SPLINE
SPL {X  -157.536, Y  +349.586, Z    +0.000, E1   +71.787, E3 +25840.740}
SPL {X  -154.855, Y  +337.291, Z    +0.000, E1   +72.155, E3 +25845.494}
SPL {X  -150.925, Y  +324.412, Z    +0.000, E1   +72.419, E3 +25851.389}
SPL {X  -146.819, Y  +313.931, Z    +0.000, E1   +72.621, E3 +25856.082}
SPL {X  -140.820, Y  +301.561, Z    +0.000, E1   +73.023, E3 +25859.998}
SPL {X  -136.475, Y  +294.006, Z    +0.000, E1   +72.670, E3 +25866.907}
SPL {X  -133.214, Y  +288.895, Z    +0.000, E1   +72.272, E3 +25872.555}
SPL {X  -129.829, Y  +284.006, Z    +0.000, E1   +71.844, E3 +25878.030}
SPL {X  -126.314, Y  +279.309, Z    +0.000, E1   +71.374, E3 +25883.322}
SPL {X  -122.705, Y  +274.834, Z    +0.000, E1   +70.869, E3 +25888.333}
SPL {X  -119.804, Y  +271.463, Z    +0.000, E1   +70.429, E3 +25892.052}
SPL {X   -77.409, Y  +237.483, Z    +0.000, E1   +59.013, E3 +25985.728}
ENDSPLINE

SPLINE
SPL {X  -103.775, Y  +255.731, Z    +0.000, E1   +56.205, E3 +26182.441}
SPL {X  -141.196, Y  +302.265, Z    +0.000, E1   +49.914, E3 +26219.926}
SPL {X  -155.405, Y  +339.473, Z    +0.000, E1   +34.418, E3 +26229.626}
SPL {X  -159.172, Y  +361.346, Z    +0.000, E1   +18.323, E3 +26232.051}
SPL {X  -159.962, Y  +374.520, Z    +0.000, E1    +5.534, E3 +26232.664}
SPL {X  -159.990, Y  +379.490, Z    +0.000, E1    +0.023, E3 +26232.721}
SPL {X  -159.990, Y  +381.667, Z    +0.000, E1    -4.707, E3 +26232.743}
SPL {X  -159.990, Y  +387.434, Z    +0.000, E1   -19.600, E3 +26232.926}
SPL {X  -159.990, Y  +395.000, Z    +0.000, E1   -38.121, E3 +26233.435}
SPL {X  -159.990, Y  +406.380, Z    +0.000, E1   -55.108, E3 +26234.876}
SPL {X  -159.990, Y  +426.664, Z    +0.000, E1   -66.963, E3 +26239.066}
SPL {X  -159.990, Y  +494.829, Z    +0.000, E1   -73.764, E3 +26260.831}
SPL {X  -158.798, Y  +695.991, Z    +0.000, E1   -74.986, E3 +26350.763}
SPL {X  -156.512, Y  +709.677, Z    +0.000, E1   -74.772, E3 +26360.907}
SPL {X  -153.684, Y  +720.975, Z    +0.000, E1   -74.508, E3 +26370.194}
SPL {X  -149.353, Y  +733.863, Z    +0.000, E1   -74.100, E3 +26381.782}
SPL {X  -145.190, Y  +743.705, Z    +0.000, E1   -73.640, E3 +26391.463}
SPL {X  -141.940, Y  +750.322, Z    +0.000, E1   -73.290, E3 +26398.230}
SPL {X  -138.555, Y  +756.496, Z    +0.000, E1   -72.905, E3 +26404.795}
SPL {X  -135.025, Y  +762.319, Z    +0.000, E1   -72.483, E3 +26411.174}
SPL {X  -131.747, Y  +767.272, Z    +0.000, E1   -72.071, E3 +26416.699}
SPL {X  -127.432, Y  +773.236, Z    +0.000, E1   -71.530, E3 +26423.385}
SPL {X  -124.036, Y  +777.554, Z    +0.000, E1   -71.026, E3 +26428.283}
SPL {X  -120.782, Y  +781.422, Z    +0.000, E1   -70.584, E3 +26432.541}
SPL {X   -74.295, Y  +818.193, Z    +0.000, E1   -57.793, E3 +26542.872}
ENDSPLINE

SPLINE
SPL {X  -105.102, Y  +797.125, Z    +0.000, E1   -55.734, E3 +26722.238}
SPL {X  -126.361, Y  +774.631, Z    +0.000, E1   -54.192, E3 +26747.906}
SPL {X  -145.777, Y  +742.423, Z    +0.000, E1   -46.722, E3 +26763.247}
SPL {X  -154.920, Y  +716.458, Z    +0.000, E1   -35.175, E3 +26769.302}
SPL {X  -159.063, Y  +693.702, Z    +0.000, E1   -19.028, E3 +26772.083}
SPL {X  -159.958, Y  +679.684, Z    +0.000, E1    -5.688, E3 +26772.795}
SPL {X  -159.990, Y  +674.512, Z    +0.000, E1    -0.026, E3 +26772.860}
SPL {X  -159.990, Y  +672.767, Z    +0.000, E1    +3.705, E3 +26772.873}
SPL {X  -159.990, Y  +669.310, Z    +0.000, E1   +12.444, E3 +26772.947}
SPL {X  -159.990, Y  +665.511, Z    +0.000, E1   +22.359, E3 +26773.106}
SPL {X  -159.990, Y  +660.776, Z    +0.000, E1   +34.018, E3 +26773.413}
SPL {X  -159.990, Y  +655.863, Z    +0.000, E1   +43.768, E3 +26773.870}
SPL {X  -159.990, Y  +646.280, Z    +0.000, E1   +56.156, E3 +26775.159}
SPL {X  -159.990, Y  +625.549, Z    +0.000, E1   +67.208, E3 +26779.681}
SPL {X  -159.990, Y  +550.186, Z    +0.000, E1   +73.637, E3 +26805.087}
SPL {X  -159.493, Y  +364.902, Z    +0.000, E1   +74.541, E3 +26892.080}
SPL {X  -156.915, Y  +346.281, Z    +0.000, E1   +74.304, E3 +26905.676}
ENDSPLINE

SPLINE
SPL {X  -159.697, Y  +367.814, Z    +0.000, E1   +71.217, E3 +26922.994}
ENDSPLINE

SPLINE
SPL {X  -157.536, Y  +349.586, Z    +0.000, E1   +71.787, E3 +26930.293}
SPL {X  -154.855, Y  +337.291, Z    +0.000, E1   +72.155, E3 +26935.047}
SPL {X  -150.925, Y  +324.412, Z    +0.000, E1   +72.419, E3 +26940.941}
SPL {X  -146.819, Y  +313.931, Z    +0.000, E1   +72.621, E3 +26945.634}
SPL {X  -140.820, Y  +301.561, Z    +0.000, E1   +73.023, E3 +26949.550}
SPL {X  -136.475, Y  +294.006, Z    +0.000, E1   +72.670, E3 +26956.459}
SPL {X  -133.214, Y  +288.895, Z    +0.000, E1   +72.272, E3 +26962.107}
SPL {X  -129.829, Y  +284.006, Z    +0.000, E1   +71.844, E3 +26967.582}
SPL {X  -126.314, Y  +279.309, Z    +0.000, E1   +71.374, E3 +26972.874}
SPL {X  -122.705, Y  +274.834, Z    +0.000, E1   +70.869, E3 +26977.886}
SPL {X  -119.804, Y  +271.463, Z    +0.000, E1   +70.429, E3 +26981.604}
SPL {X   -77.409, Y  +237.483, Z    +0.000, E1   +59.013, E3 +27075.280}
ENDSPLINE

SPLINE
SPL {X  -103.775, Y  +255.731, Z    +0.000, E1   +56.205, E3 +27271.993}
SPL {X  -141.196, Y  +302.265, Z    +0.000, E1   +49.914, E3 +27309.478}
SPL {X  -155.405, Y  +339.473, Z    +0.000, E1   +34.418, E3 +27319.179}
SPL {X  -159.172, Y  +361.346, Z    +0.000, E1   +18.323, E3 +27321.603}
SPL {X  -159.962, Y  +374.520, Z    +0.000, E1    +5.534, E3 +27322.216}
SPL {X  -159.990, Y  +379.490, Z    +0.000, E1    +0.023, E3 +27322.274}
SPL {X  -159.990, Y  +381.667, Z    +0.000, E1    -4.707, E3 +27322.295}
SPL {X  -159.990, Y  +387.434, Z    +0.000, E1   -19.600, E3 +27322.478}
SPL {X  -159.990, Y  +395.000, Z    +0.000, E1   -38.121, E3 +27322.987}
SPL {X  -159.990, Y  +406.380, Z    +0.000, E1   -55.108, E3 +27324.429}
SPL {X  -159.990, Y  +426.664, Z    +0.000, E1   -66.963, E3 +27328.619}
SPL {X  -159.990, Y  +494.829, Z    +0.000, E1   -73.764, E3 +27350.383}
SPL {X  -158.798, Y  +695.991, Z    +0.000, E1   -74.986, E3 +27440.315}
SPL {X  -156.512, Y  +709.677, Z    +0.000, E1   -74.772, E3 +27450.459}
SPL {X  -153.684, Y  +720.975, Z    +0.000, E1   -74.508, E3 +27459.746}
SPL {X  -149.353, Y  +733.863, Z    +0.000, E1   -74.100, E3 +27471.334}
SPL {X  -145.190, Y  +743.705, Z    +0.000, E1   -73.640, E3 +27481.015}
SPL {X  -141.940, Y  +750.322, Z    +0.000, E1   -73.290, E3 +27487.782}
SPL {X  -138.555, Y  +756.496, Z    +0.000, E1   -72.905, E3 +27494.347}
SPL {X  -135.025, Y  +762.319, Z    +0.000, E1   -72.483, E3 +27500.727}
SPL {X  -131.747, Y  +767.272, Z    +0.000, E1   -72.071, E3 +27506.252}
SPL {X  -127.432, Y  +773.236, Z    +0.000, E1   -71.530, E3 +27512.937}
SPL {X  -124.036, Y  +777.554, Z    +0.000, E1   -71.026, E3 +27517.835}
SPL {X  -120.782, Y  +781.422, Z    +0.000, E1   -70.584, E3 +27522.093}
SPL {X   -74.295, Y  +818.193, Z    +0.000, E1   -57.793, E3 +27632.424}
ENDSPLINE

SPLINE
SPL {X  -105.102, Y  +797.125, Z    +0.000, E1   -55.734, E3 +27811.791}
SPL {X  -126.361, Y  +774.631, Z    +0.000, E1   -54.192, E3 +27837.458}
SPL {X  -145.777, Y  +742.423, Z    +0.000, E1   -46.722, E3 +27852.799}
SPL {X  -154.920, Y  +716.458, Z    +0.000, E1   -35.175, E3 +27858.854}
SPL {X  -158.252, Y  +700.019, Z    +0.000, E1   -24.087, E3 +27861.106}
SPL {X  -159.434, Y  +689.826, Z    +0.000, E1   -15.506, E3 +27861.924}
SPL {X  -159.958, Y  +679.684, Z    +0.000, E1    -5.688, E3 +27862.347}
SPL {X  -159.990, Y  +674.512, Z    +0.000, E1    -0.026, E3 +27862.412}
SPL {X  -159.990, Y  +672.767, Z    +0.000, E1    +3.705, E3 +27862.425}
SPL {X  -159.990, Y  +669.310, Z    +0.000, E1   +12.444, E3 +27862.499}
SPL {X  -159.990, Y  +665.511, Z    +0.000, E1   +22.359, E3 +27862.658}
SPL {X  -159.990, Y  +660.776, Z    +0.000, E1   +34.018, E3 +27862.965}
SPL {X  -159.990, Y  +655.863, Z    +0.000, E1   +43.768, E3 +27863.422}
SPL {X  -159.990, Y  +646.280, Z    +0.000, E1   +56.156, E3 +27864.712}
SPL {X  -159.990, Y  +625.549, Z    +0.000, E1   +67.208, E3 +27869.233}
SPL {X  -159.990, Y  +550.186, Z    +0.000, E1   +73.637, E3 +27894.639}
SPL {X  -159.878, Y  +371.520, Z    +0.000, E1   +74.559, E3 +27977.401}
SPL {X  -159.109, Y  +360.737, Z    +0.000, E1   +74.490, E3 +27984.525}
SPL {X  -156.915, Y  +346.281, Z    +0.000, E1   +74.304, E3 +27995.228}
ENDSPLINE

SPLINE
SPL {X  -159.697, Y  +367.814, Z    +0.000, E1   +71.217, E3 +28012.547}
ENDSPLINE

SPLINE
SPL {X  -156.028, Y  +342.114, Z    +0.000, E1   +72.020, E3 +28022.700}
SPL {X  -150.925, Y  +324.412, Z    +0.000, E1   +72.419, E3 +28030.493}
SPL {X  -144.972, Y  +309.824, Z    +0.000, E1   +72.799, E3 +28036.095}
SPL {X  -139.605, Y  +299.351, Z    +0.000, E1   +73.035, E3 +28040.227}
SPL {X  -136.475, Y  +294.006, Z    +0.000, E1   +72.670, E3 +28046.012}
SPL {X  -133.214, Y  +288.895, Z    +0.000, E1   +72.272, E3 +28051.659}
SPL {X  -129.829, Y  +284.006, Z    +0.000, E1   +71.844, E3 +28057.134}
SPL {X  -126.314, Y  +279.309, Z    +0.000, E1   +71.374, E3 +28062.427}
SPL {X  -122.705, Y  +274.834, Z    +0.000, E1   +70.869, E3 +28067.438}
SPL {X  -119.804, Y  +271.463, Z    +0.000, E1   +70.429, E3 +28071.157}
SPL {X   -77.409, Y  +237.483, Z    +0.000, E1   +59.013, E3 +28164.832}
ENDSPLINE

SPLINE
SPL {X  -103.775, Y  +255.731, Z    +0.000, E1   +56.205, E3 +28361.545}
SPL {X  -133.021, Y  +288.605, Z    +0.000, E1   +53.007, E3 +28393.002}
SPL {X  -149.384, Y  +320.219, Z    +0.000, E1   +43.953, E3 +28404.725}
SPL {X  -157.534, Y  +349.577, Z    +0.000, E1   +27.748, E3 +28410.077}
SPL {X  -159.460, Y  +364.489, Z    +0.000, E1   +15.407, E3 +28411.373}
SPL {X  -159.962, Y  +374.520, Z    +0.000, E1    +5.534, E3 +28411.768}
SPL {X  -159.990, Y  +379.490, Z    +0.000, E1    +0.023, E3 +28411.826}
SPL {X  -159.990, Y  +381.667, Z    +0.000, E1    -4.707, E3 +28411.848}
SPL {X  -159.990, Y  +387.434, Z    +0.000, E1   -19.600, E3 +28412.030}
SPL {X  -159.990, Y  +392.971, Z    +0.000, E1   -33.903, E3 +28412.363}
SPL {X  -159.990, Y  +399.006, Z    +0.000, E1   -45.565, E3 +28412.939}
SPL {X  -159.990, Y  +410.008, Z    +0.000, E1   -58.546, E3 +28414.550}
SPL {X  -159.990, Y  +426.664, Z    +0.000, E1   -66.963, E3 +28418.171}
SPL {X  -159.990, Y  +494.829, Z    +0.000, E1   -73.764, E3 +28439.935}
SPL {X  -158.798, Y  +695.991, Z    +0.000, E1   -74.986, E3 +28529.868}
SPL {X  -156.512, Y  +709.677, Z    +0.000, E1   -74.772, E3 +28540.011}
SPL {X  -153.684, Y  +720.975, Z    +0.000, E1   -74.508, E3 +28549.299}
SPL {X  -149.353, Y  +733.863, Z    +0.000, E1   -74.100, E3 +28560.886}
SPL {X  -145.190, Y  +743.705, Z    +0.000, E1   -73.640, E3 +28570.567}
SPL {X  -141.940, Y  +750.322, Z    +0.000, E1   -73.290, E3 +28577.334}
SPL {X  -138.555, Y  +756.496, Z    +0.000, E1   -72.905, E3 +28583.899}
SPL {X  -135.025, Y  +762.319, Z    +0.000, E1   -72.483, E3 +28590.279}
SPL {X  -131.747, Y  +767.272, Z    +0.000, E1   -72.071, E3 +28595.804}
SPL {X  -128.648, Y  +771.613, Z    +0.000, E1   -71.666, E3 +28600.696}
SPL {X  -125.012, Y  +776.344, Z    +0.000, E1   -71.184, E3 +28606.008}
SPL {X  -121.578, Y  +780.498, Z    +0.000, E1   -70.681, E3 +28610.651}
SPL {X  -119.460, Y  +782.925, Z    +0.000, E1   -70.353, E3 +28613.315}
SPL {X   -74.295, Y  +818.193, Z    +0.000, E1   -57.793, E3 +28721.976}
ENDSPLINE

SPLINE
SPL {X  -120.240, Y  +782.043, Z    +0.000, E1   -55.019, E3 +28920.472}
SPL {X  -145.777, Y  +742.423, Z    +0.000, E1   -46.722, E3 +28942.351}
SPL {X  -154.920, Y  +716.458, Z    +0.000, E1   -35.175, E3 +28948.406}
SPL {X  -159.063, Y  +693.702, Z    +0.000, E1   -19.028, E3 +28951.188}
SPL {X  -159.958, Y  +679.684, Z    +0.000, E1    -5.688, E3 +28951.900}
SPL {X  -159.990, Y  +674.512, Z    +0.000, E1    -0.026, E3 +28951.964}
SPL {X  -159.990, Y  +672.767, Z    +0.000, E1    +3.705, E3 +28951.978}
SPL {X  -159.990, Y  +669.310, Z    +0.000, E1   +12.444, E3 +28952.052}
SPL {X  -159.990, Y  +665.511, Z    +0.000, E1   +22.359, E3 +28952.210}
SPL {X  -159.990, Y  +658.432, Z    +0.000, E1   +38.720, E3 +28952.735}
SPL {X  -159.990, Y  +646.280, Z    +0.000, E1   +56.156, E3 +28954.264}
SPL {X  -159.990, Y  +625.549, Z    +0.000, E1   +67.208, E3 +28958.785}
SPL {X  -159.990, Y  +550.186, Z    +0.000, E1   +73.637, E3 +28984.191}
SPL {X  -159.878, Y  +371.520, Z    +0.000, E1   +74.559, E3 +29066.953}
SPL {X  -159.109, Y  +360.737, Z    +0.000, E1   +74.490, E3 +29074.077}
SPL {X  -156.915, Y  +346.281, Z    +0.000, E1   +74.304, E3 +29084.780}
ENDSPLINE

SPLINE
SPL {X  -159.697, Y  +367.814, Z    +0.000, E1   +71.217, E3 +29102.099}
ENDSPLINE

SPLINE
SPL {X  -156.028, Y  +342.114, Z    +0.000, E1   +72.020, E3 +29112.252}
SPL {X  -150.925, Y  +324.412, Z    +0.000, E1   +72.419, E3 +29120.045}
SPL {X  -144.972, Y  +309.824, Z    +0.000, E1   +72.799, E3 +29125.647}
SPL {X  -139.605, Y  +299.351, Z    +0.000, E1   +73.035, E3 +29129.779}
SPL {X  -136.475, Y  +294.006, Z    +0.000, E1   +72.670, E3 +29135.564}
SPL {X  -133.214, Y  +288.895, Z    +0.000, E1   +72.272, E3 +29141.212}
SPL {X  -129.829, Y  +284.006, Z    +0.000, E1   +71.844, E3 +29146.687}
SPL {X  -126.314, Y  +279.309, Z    +0.000, E1   +71.374, E3 +29151.979}
SPL {X  -122.705, Y  +274.834, Z    +0.000, E1   +70.869, E3 +29156.990}
SPL {X  -119.804, Y  +271.463, Z    +0.000, E1   +70.429, E3 +29160.709}
SPL {X   -77.409, Y  +237.483, Z    +0.000, E1   +59.013, E3 +29254.384}
ENDSPLINE

SPLINE
SPL {X  -103.775, Y  +255.731, Z    +0.000, E1   +56.205, E3 +29451.098}
SPL {X  -141.196, Y  +302.265, Z    +0.000, E1   +49.914, E3 +29488.583}
SPL {X  -155.405, Y  +339.473, Z    +0.000, E1   +34.418, E3 +29498.283}
SPL {X  -159.172, Y  +361.346, Z    +0.000, E1   +18.323, E3 +29500.708}
SPL {X  -159.962, Y  +374.520, Z    +0.000, E1    +5.534, E3 +29501.321}
SPL {X  -159.990, Y  +379.490, Z    +0.000, E1    +0.023, E3 +29501.378}
SPL {X  -159.990, Y  +381.667, Z    +0.000, E1    -4.707, E3 +29501.400}
SPL {X  -159.990, Y  +385.814, Z    +0.000, E1   -15.621, E3 +29501.504}
SPL {X  -159.990, Y  +390.948, Z    +0.000, E1   -28.850, E3 +29501.780}
SPL {X  -159.990, Y  +399.006, Z    +0.000, E1   -45.565, E3 +29502.492}
SPL {X  -159.990, Y  +410.008, Z    +0.000, E1   -58.546, E3 +29504.102}
SPL {X  -159.990, Y  +426.664, Z    +0.000, E1   -66.963, E3 +29507.723}
SPL {X  -159.990, Y  +494.829, Z    +0.000, E1   -73.764, E3 +29529.487}
SPL {X  -158.798, Y  +695.991, Z    +0.000, E1   -74.986, E3 +29619.420}
SPL {X  -156.512, Y  +709.677, Z    +0.000, E1   -74.772, E3 +29629.564}
SPL {X  -153.684, Y  +720.975, Z    +0.000, E1   -74.508, E3 +29638.851}
SPL {X  -149.353, Y  +733.863, Z    +0.000, E1   -74.100, E3 +29650.439}
SPL {X  -145.190, Y  +743.705, Z    +0.000, E1   -73.640, E3 +29660.120}
SPL {X  -141.940, Y  +750.322, Z    +0.000, E1   -73.290, E3 +29666.887}
SPL {X  -138.555, Y  +756.496, Z    +0.000, E1   -72.905, E3 +29673.452}
SPL {X  -135.025, Y  +762.319, Z    +0.000, E1   -72.483, E3 +29679.831}
SPL {X  -131.747, Y  +767.272, Z    +0.000, E1   -72.071, E3 +29685.356}
SPL {X  -128.648, Y  +771.613, Z    +0.000, E1   -71.666, E3 +29690.248}
SPL {X  -125.012, Y  +776.344, Z    +0.000, E1   -71.184, E3 +29695.560}
SPL {X  -120.782, Y  +781.422, Z    +0.000, E1   -70.584, E3 +29701.198}
SPL {X   -74.295, Y  +818.193, Z    +0.000, E1   -57.793, E3 +29811.528}
ENDSPLINE

SPLINE
SPL {X  -120.240, Y  +782.043, Z    +0.000, E1   -55.019, E3 +30010.024}
SPL {X  -145.777, Y  +742.423, Z    +0.000, E1   -46.722, E3 +30031.904}
SPL {X  -154.920, Y  +716.458, Z    +0.000, E1   -35.175, E3 +30037.959}
SPL {X  -158.252, Y  +700.019, Z    +0.000, E1   -24.087, E3 +30040.210}
SPL {X  -159.676, Y  +686.525, Z    +0.000, E1   -12.514, E3 +30041.200}
SPL {X  -159.990, Y  +674.678, Z    +0.000, E1    -0.382, E3 +30041.515}
SPL {X  -159.990, Y  +672.767, Z    +0.000, E1    +3.705, E3 +30041.530}
SPL {X  -159.990, Y  +669.310, Z    +0.000, E1   +12.444, E3 +30041.604}
SPL {X  -159.990, Y  +665.511, Z    +0.000, E1   +22.359, E3 +30041.763}
SPL {X  -159.990, Y  +660.776, Z    +0.000, E1   +34.018, E3 +30042.069}
SPL {X  -159.990, Y  +655.863, Z    +0.000, E1   +43.768, E3 +30042.527}
SPL {X  -159.990, Y  +646.280, Z    +0.000, E1   +56.156, E3 +30043.816}
SPL {X  -159.990, Y  +625.549, Z    +0.000, E1   +67.208, E3 +30048.338}
SPL {X  -159.990, Y  +550.186, Z    +0.000, E1   +73.637, E3 +30073.743}
SPL {X  -159.493, Y  +364.902, Z    +0.000, E1   +74.541, E3 +30160.737}
SPL {X  -156.915, Y  +346.281, Z    +0.000, E1   +74.304, E3 +30174.333}
ENDSPLINE

SPLINE
SPL {X  -159.697, Y  +367.814, Z    +0.000, E1   +71.217, E3 +30191.651}
ENDSPLINE

SPLINE
SPL {X  -157.536, Y  +349.586, Z    +0.000, E1   +71.787, E3 +30198.949}
SPL {X  -154.855, Y  +337.291, Z    +0.000, E1   +72.155, E3 +30203.703}
SPL {X  -150.925, Y  +324.412, Z    +0.000, E1   +72.419, E3 +30209.598}
SPL {X  -144.972, Y  +309.824, Z    +0.000, E1   +72.799, E3 +30215.200}
SPL {X  -139.605, Y  +299.351, Z    +0.000, E1   +73.035, E3 +30219.331}
SPL {X  -136.475, Y  +294.006, Z    +0.000, E1   +72.670, E3 +30225.116}
SPL {X  -133.214, Y  +288.895, Z    +0.000, E1   +72.272, E3 +30230.764}
SPL {X  -129.829, Y  +284.006, Z    +0.000, E1   +71.844, E3 +30236.239}
SPL {X  -125.428, Y  +278.179, Z    +0.000, E1   +71.273, E3 +30242.776}
SPL {X  -120.729, Y  +272.518, Z    +0.000, E1   +70.593, E3 +30249.086}
SPL {X   -77.409, Y  +237.483, Z    +0.000, E1   +59.013, E3 +30343.937}
ENDSPLINE

SPLINE
SPL {X  -103.775, Y  +255.731, Z    +0.000, E1   +56.205, E3 +30540.650}
SPL {X  -141.196, Y  +302.265, Z    +0.000, E1   +49.914, E3 +30578.135}
SPL {X  -155.405, Y  +339.473, Z    +0.000, E1   +34.418, E3 +30587.835}
SPL {X  -159.172, Y  +361.346, Z    +0.000, E1   +18.323, E3 +30590.260}
SPL {X  -159.962, Y  +374.520, Z    +0.000, E1    +5.534, E3 +30590.873}
SPL {X  -159.990, Y  +379.741, Z    +0.000, E1    -0.257, E3 +30590.932}
SPL {X  -159.990, Y  +384.604, Z    +0.000, E1   -12.124, E3 +30591.020}
SPL {X  -159.990, Y  +389.475, Z    +0.000, E1   -25.351, E3 +30591.234}
SPL {X  -159.990, Y  +395.000, Z    +0.000, E1   -38.121, E3 +30591.644}
SPL {X  -159.990, Y  +406.380, Z    +0.000, E1   -55.108, E3 +30593.085}
SPL {X  -159.990, Y  +426.664, Z    +0.000, E1   -66.963, E3 +30597.275}
SPL {X  -159.990, Y  +494.829, Z    +0.000, E1   -73.764, E3 +30619.040}
SPL {X  -158.798, Y  +695.991, Z    +0.000, E1   -74.986, E3 +30708.972}
SPL {X  -156.512, Y  +709.677, Z    +0.000, E1   -74.772, E3 +30719.116}
SPL {X  -153.684, Y  +720.975, Z    +0.000, E1   -74.508, E3 +30728.403}
SPL {X  -149.353, Y  +733.863, Z    +0.000, E1   -74.100, E3 +30739.991}
SPL {X  -145.190, Y  +743.705, Z    +0.000, E1   -73.640, E3 +30749.672}
SPL {X  -141.940, Y  +750.322, Z    +0.000, E1   -73.290, E3 +30756.439}
SPL {X  -138.555, Y  +756.496, Z    +0.000, E1   -72.905, E3 +30763.004}
SPL {X  -135.025, Y  +762.319, Z    +0.000, E1   -72.483, E3 +30769.383}
SPL {X  -131.747, Y  +767.272, Z    +0.000, E1   -72.071, E3 +30774.908}
SPL {X  -127.432, Y  +773.236, Z    +0.000, E1   -71.530, E3 +30781.594}
SPL {X  -124.036, Y  +777.554, Z    +0.000, E1   -71.026, E3 +30786.492}
SPL {X  -120.782, Y  +781.422, Z    +0.000, E1   -70.584, E3 +30790.750}
SPL {X   -74.295, Y  +818.193, Z    +0.000, E1   -57.793, E3 +30901.081}
ENDSPLINE

SPLINE
SPL {X  -120.240, Y  +782.043, Z    +0.000, E1   -55.019, E3 +31099.577}
SPL {X  -145.777, Y  +742.423, Z    +0.000, E1   -46.722, E3 +31121.456}
SPL {X  -154.920, Y  +716.458, Z    +0.000, E1   -35.175, E3 +31127.511}
SPL {X  -159.063, Y  +693.702, Z    +0.000, E1   -19.028, E3 +31130.292}
SPL {X  -159.958, Y  +679.684, Z    +0.000, E1    -5.688, E3 +31131.004}
SPL {X  -159.990, Y  +674.512, Z    +0.000, E1    -0.026, E3 +31131.069}
SPL {X  -159.990, Y  +672.767, Z    +0.000, E1    +3.705, E3 +31131.082}
SPL {X  -159.990, Y  +669.310, Z    +0.000, E1   +12.444, E3 +31131.156}
SPL {X  -159.990, Y  +665.511, Z    +0.000, E1   +22.359, E3 +31131.315}
SPL {X  -159.990, Y  +658.432, Z    +0.000, E1   +38.720, E3 +31131.840}
SPL {X  -159.990, Y  +646.280, Z    +0.000, E1   +56.156, E3 +31133.368}
SPL {X  -159.990, Y  +625.549, Z    +0.000, E1   +67.208, E3 +31137.890}
SPL {X  -159.990, Y  +550.186, Z    +0.000, E1   +73.637, E3 +31163.296}
SPL {X  -159.493, Y  +364.902, Z    +0.000, E1   +74.541, E3 +31250.289}
SPL {X  -156.915, Y  +346.281, Z    +0.000, E1   +74.304, E3 +31263.885}
ENDSPLINE

SPLINE
SPL {X  -159.697, Y  +367.814, Z    +0.000, E1   +71.217, E3 +31281.203}
ENDSPLINE

SPLINE
SPL {X  -157.536, Y  +349.586, Z    +0.000, E1   +71.787, E3 +31288.501}
SPL {X  -154.855, Y  +337.291, Z    +0.000, E1   +72.155, E3 +31293.256}
SPL {X  -150.925, Y  +324.412, Z    +0.000, E1   +72.419, E3 +31299.150}
SPL {X  -144.972, Y  +309.824, Z    +0.000, E1   +72.799, E3 +31304.752}
SPL {X  -139.605, Y  +299.351, Z    +0.000, E1   +73.035, E3 +31308.883}
SPL {X  -136.475, Y  +294.006, Z    +0.000, E1   +72.670, E3 +31314.668}
SPL {X  -133.214, Y  +288.895, Z    +0.000, E1   +72.272, E3 +31320.316}
SPL {X  -129.829, Y  +284.006, Z    +0.000, E1   +71.844, E3 +31325.791}
SPL {X  -126.314, Y  +279.309, Z    +0.000, E1   +71.374, E3 +31331.083}
SPL {X  -122.705, Y  +274.834, Z    +0.000, E1   +70.869, E3 +31336.095}
SPL {X  -119.804, Y  +271.463, Z    +0.000, E1   +70.429, E3 +31339.813}
SPL {X   -77.409, Y  +237.483, Z    +0.000, E1   +59.013, E3 +31433.489}
ENDSPLINE

SPLINE
SPL {X  -103.775, Y  +255.731, Z    +0.000, E1   +56.205, E3 +31630.202}
SPL {X  -141.196, Y  +302.265, Z    +0.000, E1   +49.914, E3 +31667.687}
SPL {X  -155.405, Y  +339.473, Z    +0.000, E1   +34.418, E3 +31677.388}
SPL {X  -159.172, Y  +361.346, Z    +0.000, E1   +18.323, E3 +31679.812}
SPL {X  -159.962, Y  +374.520, Z    +0.000, E1    +5.534, E3 +31680.425}
SPL {X  -159.990, Y  +379.490, Z    +0.000, E1    +0.023, E3 +31680.483}
SPL {X  -159.990, Y  +381.667, Z    +0.000, E1    -4.707, E3 +31680.504}
SPL {X  -159.990, Y  +385.814, Z    +0.000, E1   -15.621, E3 +31680.608}
SPL {X  -159.990, Y  +390.948, Z    +0.000, E1   -28.850, E3 +31680.885}
SPL {X  -159.990, Y  +399.006, Z    +0.000, E1   -45.565, E3 +31681.596}
SPL {X  -159.990, Y  +410.008, Z    +0.000, E1   -58.546, E3 +31683.207}
SPL {X  -159.990, Y  +426.664, Z    +0.000, E1   -66.963, E3 +31686.828}
SPL {X  -159.990, Y  +494.829, Z    +0.000, E1   -73.764, E3 +31708.592}
SPL {X  -158.798, Y  +695.991, Z    +0.000, E1   -74.986, E3 +31798.524}
SPL {X  -156.512, Y  +709.677, Z    +0.000, E1   -74.772, E3 +31808.668}
SPL {X  -153.684, Y  +720.975, Z    +0.000, E1   -74.508, E3 +31817.955}
SPL {X  -149.353, Y  +733.863, Z    +0.000, E1   -74.100, E3 +31829.543}
SPL {X  -145.190, Y  +743.705, Z    +0.000, E1   -73.640, E3 +31839.224}
SPL {X  -141.940, Y  +750.322, Z    +0.000, E1   -73.290, E3 +31845.991}
SPL {X  -138.555, Y  +756.496, Z    +0.000, E1   -72.905, E3 +31852.556}
SPL {X  -135.025, Y  +762.319, Z    +0.000, E1   -72.483, E3 +31858.936}
SPL {X  -131.747, Y  +767.272, Z    +0.000, E1   -72.071, E3 +31864.461}
SPL {X  -127.432, Y  +773.236, Z    +0.000, E1   -71.530, E3 +31871.146}
SPL {X  -122.390, Y  +779.541, Z    +0.000, E1   -70.825, E3 +31878.221}
SPL {X  -119.460, Y  +782.925, Z    +0.000, E1   -70.353, E3 +31881.972}
SPL {X   -74.295, Y  +818.193, Z    +0.000, E1   -57.793, E3 +31990.633}
ENDSPLINE

SPLINE
SPL {X  -120.240, Y  +782.043, Z    +0.000, E1   -55.019, E3 +32189.129}
SPL {X  -145.777, Y  +742.423, Z    +0.000, E1   -46.722, E3 +32211.008}
SPL {X  -154.920, Y  +716.458, Z    +0.000, E1   -35.175, E3 +32217.063}
SPL {X  -158.252, Y  +700.019, Z    +0.000, E1   -24.087, E3 +32219.315}
SPL {X  -159.434, Y  +689.826, Z    +0.000, E1   -15.506, E3 +32220.133}
SPL {X  -159.958, Y  +679.684, Z    +0.000, E1    -5.688, E3 +32220.556}
SPL {X  -159.990, Y  +674.512, Z    +0.000, E1    -0.026, E3 +32220.621}
SPL {X  -159.990, Y  +672.767, Z    +0.000, E1    +3.705, E3 +32220.634}
SPL {X  -159.990, Y  +669.310, Z    +0.000, E1   +12.444, E3 +32220.708}
SPL {X  -159.990, Y  +665.511, Z    +0.000, E1   +22.359, E3 +32220.867}
SPL {X  -159.990, Y  +658.432, Z    +0.000, E1   +38.720, E3 +32221.392}
SPL {X  -159.990, Y  +646.280, Z    +0.000, E1   +56.156, E3 +32222.920}
SPL {X  -159.990, Y  +625.549, Z    +0.000, E1   +67.208, E3 +32227.442}
SPL {X  -159.990, Y  +550.186, Z    +0.000, E1   +73.637, E3 +32252.848}
SPL {X  -159.493, Y  +364.902, Z    +0.000, E1   +74.541, E3 +32339.841}
SPL {X  -156.915, Y  +346.281, Z    +0.000, E1   +74.304, E3 +32353.437}
ENDSPLINE

SPLINE
SPL {X  -159.697, Y  +367.814, Z    +0.000, E1   +71.217, E3 +32370.756}
ENDSPLINE

SPLINE
SPL {X  -156.028, Y  +342.114, Z    +0.000, E1   +72.020, E3 +32380.909}
SPL {X  -150.925, Y  +324.412, Z    +0.000, E1   +72.419, E3 +32388.702}
SPL {X  -144.972, Y  +309.824, Z    +0.000, E1   +72.799, E3 +32394.304}
SPL {X  -139.605, Y  +299.351, Z    +0.000, E1   +73.035, E3 +32398.436}
SPL {X  -136.475, Y  +294.006, Z    +0.000, E1   +72.670, E3 +32404.221}
SPL {X  -133.214, Y  +288.895, Z    +0.000, E1   +72.272, E3 +32409.868}
SPL {X  -129.829, Y  +284.006, Z    +0.000, E1   +71.844, E3 +32415.343}
SPL {X  -125.428, Y  +278.179, Z    +0.000, E1   +71.273, E3 +32421.881}
SPL {X  -120.729, Y  +272.518, Z    +0.000, E1   +70.593, E3 +32428.190}
SPL {X   -77.409, Y  +237.483, Z    +0.000, E1   +59.013, E3 +32523.041}
ENDSPLINE

SPLINE
SPL {X  -103.775, Y  +255.731, Z    +0.000, E1   +56.205, E3 +32719.754}
SPL {X  -141.196, Y  +302.265, Z    +0.000, E1   +49.914, E3 +32757.239}
SPL {X  -153.296, Y  +331.706, Z    +0.000, E1   +38.681, E3 +32765.658}
SPL {X  -157.534, Y  +349.577, Z    +0.000, E1   +27.748, E3 +32768.286}
SPL {X  -159.460, Y  +364.489, Z    +0.000, E1   +15.407, E3 +32769.582}
SPL {X  -159.962, Y  +374.520, Z    +0.000, E1    +5.534, E3 +32769.977}
SPL {X  -159.990, Y  +379.490, Z    +0.000, E1    +0.023, E3 +32770.035}
SPL {X  -159.990, Y  +381.667, Z    +0.000, E1    -4.707, E3 +32770.057}
SPL {X  -159.990, Y  +385.814, Z    +0.000, E1   -15.621, E3 +32770.161}
SPL {X  -159.990, Y  +390.948, Z    +0.000, E1   -28.850, E3 +32770.437}
SPL {X  -159.990, Y  +399.006, Z    +0.000, E1   -45.565, E3 +32771.148}
SPL {X  -159.990, Y  +410.008, Z    +0.000, E1   -58.546, E3 +32772.759}
SPL {X  -159.990, Y  +430.714, Z    +0.000, E1   -67.965, E3 +32777.564}
SPL {X  -159.990, Y  +500.758, Z    +0.000, E1   -73.927, E3 +32800.240}
SPL {X  -158.798, Y  +695.991, Z    +0.000, E1   -74.986, E3 +32888.077}
SPL {X  -156.512, Y  +709.677, Z    +0.000, E1   -74.772, E3 +32898.220}
SPL {X  -153.684, Y  +720.975, Z    +0.000, E1   -74.508, E3 +32907.508}
SPL {X  -150.879, Y  +729.719, Z    +0.000, E1   -74.224, E3 +32915.301}
SPL {X  -148.237, Y  +736.689, Z    +0.000, E1   -73.960, E3 +32921.855}
SPL {X  -145.190, Y  +743.705, Z    +0.000, E1   -73.640, E3 +32928.776}
SPL {X  -141.940, Y  +750.322, Z    +0.000, E1   -73.290, E3 +32935.543}
SPL {X  -138.555, Y  +756.496, Z    +0.000, E1   -72.905, E3 +32942.108}
SPL {X  -135.025, Y  +762.319, Z    +0.000, E1   -72.483, E3 +32948.488}
SPL {X  -131.747, Y  +767.272, Z    +0.000, E1   -72.071, E3 +32954.013}
SPL {X  -128.648, Y  +771.613, Z    +0.000, E1   -71.666, E3 +32958.905}
SPL {X  -125.012, Y  +776.344, Z    +0.000, E1   -71.184, E3 +32964.217}
SPL {X  -120.782, Y  +781.422, Z    +0.000, E1   -70.584, E3 +32969.855}
SPL {X   -74.295, Y  +818.193, Z    +0.000, E1   -57.793, E3 +33080.185}
ENDSPLINE

SPLINE
SPL {X  -120.240, Y  +782.043, Z    +0.000, E1   -55.019, E3 +33278.681}
SPL {X  -145.777, Y  +742.423, Z    +0.000, E1   -46.722, E3 +33300.560}
SPL {X  -154.920, Y  +716.458, Z    +0.000, E1   -35.175, E3 +33306.615}
SPL {X  -158.252, Y  +700.019, Z    +0.000, E1   -24.087, E3 +33308.867}
SPL {X  -159.676, Y  +686.525, Z    +0.000, E1   -12.514, E3 +33309.857}
SPL {X  -159.990, Y  +674.678, Z    +0.000, E1    -0.382, E3 +33310.172}
SPL {X  -159.990, Y  +672.767, Z    +0.000, E1    +3.705, E3 +33310.187}
SPL {X  -159.990, Y  +669.310, Z    +0.000, E1   +12.444, E3 +33310.261}
SPL {X  -159.990, Y  +665.511, Z    +0.000, E1   +22.359, E3 +33310.419}
SPL {X  -159.990, Y  +660.776, Z    +0.000, E1   +34.018, E3 +33310.726}
SPL {X  -159.990, Y  +655.863, Z    +0.000, E1   +43.768, E3 +33311.183}
SPL {X  -159.990, Y  +646.280, Z    +0.000, E1   +56.156, E3 +33312.473}
SPL {X  -159.990, Y  +625.549, Z    +0.000, E1   +67.208, E3 +33316.994}
SPL {X  -159.990, Y  +550.186, Z    +0.000, E1   +73.637, E3 +33342.400}
SPL {X  -159.878, Y  +371.520, Z    +0.000, E1   +74.559, E3 +33425.162}
SPL {X  -159.109, Y  +360.737, Z    +0.000, E1   +74.490, E3 +33432.286}
SPL {X  -156.915, Y  +346.281, Z    +0.000, E1   +74.304, E3 +33442.989}
ENDSPLINE

SPLINE
SPL {X  -159.697, Y  +367.814, Z    +0.000, E1   +71.217, E3 +33460.308}
ENDSPLINE

SPLINE
SPL {X  -156.028, Y  +342.114, Z    +0.000, E1   +72.020, E3 +33470.461}
SPL {X  -150.925, Y  +324.412, Z    +0.000, E1   +72.419, E3 +33478.254}
SPL {X  -144.972, Y  +309.824, Z    +0.000, E1   +72.799, E3 +33483.856}
SPL {X  -139.605, Y  +299.351, Z    +0.000, E1   +73.035, E3 +33487.988}
SPL {X  -136.475, Y  +294.006, Z    +0.000, E1   +72.670, E3 +33493.773}
SPL {X  -133.214, Y  +288.895, Z    +0.000, E1   +72.272, E3 +33499.421}
SPL {X  -129.829, Y  +284.006, Z    +0.000, E1   +71.844, E3 +33504.895}
SPL {X  -125.428, Y  +278.179, Z    +0.000, E1   +71.273, E3 +33511.433}
SPL {X  -120.729, Y  +272.518, Z    +0.000, E1   +70.593, E3 +33517.742}
SPL {X   -77.409, Y  +237.483, Z    +0.000, E1   +59.013, E3 +33612.593}
ENDSPLINE

SPLINE
SPL {X  -103.775, Y  +255.731, Z    +0.000, E1   +56.205, E3 +33809.307}
SPL {X  -141.196, Y  +302.265, Z    +0.000, E1   +49.914, E3 +33846.792}
SPL {X  -155.405, Y  +339.473, Z    +0.000, E1   +34.418, E3 +33856.492}
SPL {X  -159.172, Y  +361.346, Z    +0.000, E1   +18.323, E3 +33858.917}
SPL {X  -159.962, Y  +374.520, Z    +0.000, E1    +5.534, E3 +33859.530}
SPL {X  -159.990, Y  +379.490, Z    +0.000, E1    +0.023, E3 +33859.587}
SPL {X  -159.990, Y  +381.667, Z    +0.000, E1    -4.707, E3 +33859.609}
SPL {X  -159.990, Y  +385.814, Z    +0.000, E1   -15.621, E3 +33859.713}
SPL {X  -159.990, Y  +390.948, Z    +0.000, E1   -28.850, E3 +33859.989}
SPL {X  -159.990, Y  +399.006, Z    +0.000, E1   -45.565, E3 +33860.701}
SPL {X  -159.990, Y  +410.008, Z    +0.000, E1   -58.546, E3 +33862.311}
SPL {X  -159.990, Y  +426.664, Z    +0.000, E1   -66.963, E3 +33865.932}
SPL {X  -159.990, Y  +494.829, Z    +0.000, E1   -73.764, E3 +33887.696}
SPL {X  -158.798, Y  +695.991, Z    +0.000, E1   -74.986, E3 +33977.629}
SPL {X  -156.512, Y  +709.677, Z    +0.000, E1   -74.772, E3 +33987.772}
SPL {X  -153.684, Y  +720.975, Z    +0.000, E1   -74.508, E3 +33997.060}
SPL {X  -149.353, Y  +733.863, Z    +0.000, E1   -74.100, E3 +34008.648}
SPL {X  -145.190, Y  +743.705, Z    +0.000, E1   -73.640, E3 +34018.329}
SPL {X  -141.940, Y  +750.322, Z    +0.000, E1   -73.290, E3 +34025.096}
SPL {X  -138.555, Y  +756.496, Z    +0.000, E1   -72.905, E3 +34031.660}
SPL {X  -135.025, Y  +762.319, Z    +0.000, E1   -72.483, E3 +34038.040}
SPL {X  -131.747, Y  +767.272, Z    +0.000, E1   -72.071, E3 +34043.565}
SPL {X  -127.432, Y  +773.236, Z    +0.000, E1   -71.530, E3 +34050.250}
SPL {X  -124.036, Y  +777.554, Z    +0.000, E1   -71.026, E3 +34055.149}
SPL {X  -120.782, Y  +781.422, Z    +0.000, E1   -70.584, E3 +34059.407}
SPL {X   -74.295, Y  +818.193, Z    +0.000, E1   -57.793, E3 +34169.737}
ENDSPLINE

SPLINE
SPL {X  -105.102, Y  +797.125, Z    +0.000, E1   -55.734, E3 +34349.104}
SPL {X  -126.361, Y  +774.631, Z    +0.000, E1   -54.192, E3 +34374.772}
SPL {X  -145.777, Y  +742.423, Z    +0.000, E1   -46.722, E3 +34390.113}
SPL {X  -154.920, Y  +716.458, Z    +0.000, E1   -35.175, E3 +34396.168}
SPL {X  -158.252, Y  +700.019, Z    +0.000, E1   -24.087, E3 +34398.419}
SPL {X  -159.434, Y  +689.826, Z    +0.000, E1   -15.506, E3 +34399.238}
SPL {X  -159.958, Y  +679.684, Z    +0.000, E1    -5.688, E3 +34399.661}
SPL {X  -159.990, Y  +674.512, Z    +0.000, E1    -0.026, E3 +34399.726}
SPL {X  -159.990, Y  +672.767, Z    +0.000, E1    +3.705, E3 +34399.739}
SPL {X  -159.990, Y  +669.310, Z    +0.000, E1   +12.444, E3 +34399.813}
SPL {X  -159.990, Y  +665.511, Z    +0.000, E1   +22.359, E3 +34399.972}
SPL {X  -159.990, Y  +660.776, Z    +0.000, E1   +34.018, E3 +34400.278}
SPL {X  -159.990, Y  +655.863, Z    +0.000, E1   +43.768, E3 +34400.736}
SPL {X  -159.990, Y  +646.280, Z    +0.000, E1   +56.156, E3 +34402.025}
SPL {X  -159.990, Y  +625.549, Z    +0.000, E1   +67.208, E3 +34406.547}
SPL {X  -159.990, Y  +550.186, Z    +0.000, E1   +73.637, E3 +34431.952}
SPL {X  -159.878, Y  +371.520, Z    +0.000, E1   +74.559, E3 +34514.714}
SPL {X  -159.109, Y  +360.737, Z    +0.000, E1   +74.490, E3 +34521.839}
SPL {X  -156.915, Y  +346.281, Z    +0.000, E1   +74.304, E3 +34532.542}
ENDSPLINE

SPLINE
SPL {X  -159.697, Y  +367.814, Z    +0.000, E1   +71.217, E3 +34549.860}
ENDSPLINE

SPLINE
SPL {X  -157.536, Y  +349.586, Z    +0.000, E1   +71.787, E3 +34557.158}
SPL {X  -154.855, Y  +337.291, Z    +0.000, E1   +72.155, E3 +34561.912}
SPL {X  -150.925, Y  +324.412, Z    +0.000, E1   +72.419, E3 +34567.806}
SPL {X  -146.819, Y  +313.931, Z    +0.000, E1   +72.621, E3 +34572.500}
SPL {X  -140.820, Y  +301.561, Z    +0.000, E1   +73.023, E3 +34576.416}
SPL {X  -136.475, Y  +294.006, Z    +0.000, E1   +72.670, E3 +34583.325}
SPL {X  -133.214, Y  +288.895, Z    +0.000, E1   +72.272, E3 +34588.973}
SPL {X  -129.829, Y  +284.006, Z    +0.000, E1   +71.844, E3 +34594.448}
SPL {X  -126.314, Y  +279.309, Z    +0.000, E1   +71.374, E3 +34599.740}
SPL {X  -122.705, Y  +274.834, Z    +0.000, E1   +70.869, E3 +34604.751}
SPL {X  -119.804, Y  +271.463, Z    +0.000, E1   +70.429, E3 +34608.470}
SPL {X   -77.409, Y  +237.483, Z    +0.000, E1   +59.013, E3 +34702.146}
ENDSPLINE

SPLINE
SPL {X  -103.775, Y  +255.731, Z    +0.000, E1   +56.205, E3 +34898.859}
SPL {X  -141.196, Y  +302.265, Z    +0.000, E1   +49.914, E3 +34936.344}
SPL {X  -155.405, Y  +339.473, Z    +0.000, E1   +34.418, E3 +34946.044}
SPL {X  -159.172, Y  +361.346, Z    +0.000, E1   +18.323, E3 +34948.469}
SPL {X  -159.962, Y  +374.520, Z    +0.000, E1    +5.534, E3 +34949.082}
SPL {X  -159.990, Y  +379.490, Z    +0.000, E1    +0.023, E3 +34949.139}
SPL {X  -159.990, Y  +381.667, Z    +0.000, E1    -4.707, E3 +34949.161}
SPL {X  -159.990, Y  +385.814, Z    +0.000, E1   -15.621, E3 +34949.265}
SPL {X  -159.990, Y  +390.948, Z    +0.000, E1   -28.850, E3 +34949.541}
SPL {X  -159.990, Y  +399.006, Z    +0.000, E1   -45.565, E3 +34950.253}
SPL {X  -159.990, Y  +410.008, Z    +0.000, E1   -58.546, E3 +34951.863}
SPL {X  -159.990, Y  +426.664, Z    +0.000, E1   -66.963, E3 +34955.484}
SPL {X  -159.990, Y  +494.829, Z    +0.000, E1   -73.764, E3 +34977.248}
SPL {X  -158.798, Y  +695.991, Z    +0.000, E1   -74.986, E3 +35067.181}
SPL {X  -156.512, Y  +709.677, Z    +0.000, E1   -74.772, E3 +35077.325}
SPL {X  -153.684, Y  +720.975, Z    +0.000, E1   -74.508, E3 +35086.612}
SPL {X  -149.353, Y  +733.863, Z    +0.000, E1   -74.100, E3 +35098.200}
SPL {X  -145.190, Y  +743.705, Z    +0.000, E1   -73.640, E3 +35107.881}
SPL {X  -141.940, Y  +750.322, Z    +0.000, E1   -73.290, E3 +35114.648}
SPL {X  -138.555, Y  +756.496, Z    +0.000, E1   -72.905, E3 +35121.213}
SPL {X  -135.025, Y  +762.319, Z    +0.000, E1   -72.483, E3 +35127.592}
SPL {X  -131.747, Y  +767.272, Z    +0.000, E1   -72.071, E3 +35133.117}
SPL {X  -127.432, Y  +773.236, Z    +0.000, E1   -71.530, E3 +35139.803}
SPL {X  -122.390, Y  +779.541, Z    +0.000, E1   -70.825, E3 +35146.877}
SPL {X  -119.460, Y  +782.925, Z    +0.000, E1   -70.353, E3 +35150.629}
SPL {X   -74.295, Y  +818.193, Z    +0.000, E1   -57.793, E3 +35259.290}
ENDSPLINE

SPLINE
SPL {X  -120.240, Y  +782.043, Z    +0.000, E1   -55.019, E3 +35457.786}
SPL {X  -145.777, Y  +742.423, Z    +0.000, E1   -46.722, E3 +35479.665}
SPL {X  -154.920, Y  +716.458, Z    +0.000, E1   -35.175, E3 +35485.720}
SPL {X  -158.252, Y  +700.019, Z    +0.000, E1   -24.087, E3 +35487.972}
SPL {X  -159.434, Y  +689.826, Z    +0.000, E1   -15.506, E3 +35488.790}
SPL {X  -159.958, Y  +679.684, Z    +0.000, E1    -5.688, E3 +35489.213}
SPL {X  -159.990, Y  +674.512, Z    +0.000, E1    -0.026, E3 +35489.278}
SPL {X  -159.990, Y  +672.767, Z    +0.000, E1    +3.705, E3 +35489.291}
SPL {X  -159.990, Y  +669.310, Z    +0.000, E1   +12.444, E3 +35489.365}
SPL {X  -159.990, Y  +665.511, Z    +0.000, E1   +22.359, E3 +35489.524}
SPL {X  -159.990, Y  +658.432, Z    +0.000, E1   +38.720, E3 +35490.049}
SPL {X  -159.990, Y  +646.280, Z    +0.000, E1   +56.156, E3 +35491.577}
SPL {X  -159.990, Y  +625.549, Z    +0.000, E1   +67.208, E3 +35496.099}
SPL {X  -159.990, Y  +550.186, Z    +0.000, E1   +73.637, E3 +35521.505}
SPL {X  -159.493, Y  +364.902, Z    +0.000, E1   +74.541, E3 +35608.498}
SPL {X  -156.915, Y  +346.281, Z    +0.000, E1   +74.304, E3 +35622.094}
ENDSPLINE

SPLINE
SPL {X  -159.697, Y  +367.814, Z    +0.000, E1   +71.217, E3 +35639.412}
ENDSPLINE

SPLINE
SPL {X  -156.028, Y  +342.114, Z    +0.000, E1   +72.020, E3 +35649.566}
SPL {X  -150.925, Y  +324.412, Z    +0.000, E1   +72.419, E3 +35657.359}
SPL {X  -144.972, Y  +309.824, Z    +0.000, E1   +72.799, E3 +35662.961}
SPL {X  -139.605, Y  +299.351, Z    +0.000, E1   +73.035, E3 +35667.092}
SPL {X  -136.475, Y  +294.006, Z    +0.000, E1   +72.670, E3 +35672.877}
SPL {X  -133.214, Y  +288.895, Z    +0.000, E1   +72.272, E3 +35678.525}
SPL {X  -129.829, Y  +284.006, Z    +0.000, E1   +71.844, E3 +35684.000}
SPL {X  -125.428, Y  +278.179, Z    +0.000, E1   +71.273, E3 +35690.537}
SPL {X  -120.729, Y  +272.518, Z    +0.000, E1   +70.593, E3 +35696.847}
SPL {X   -77.409, Y  +237.483, Z    +0.000, E1   +59.013, E3 +35791.698}
ENDSPLINE

SPLINE
SPL {X  -103.775, Y  +255.731, Z    +0.000, E1   +56.205, E3 +35988.411}
SPL {X  -141.196, Y  +302.265, Z    +0.000, E1   +49.914, E3 +36025.896}
SPL {X  -153.296, Y  +331.706, Z    +0.000, E1   +38.681, E3 +36034.315}
SPL {X  -157.534, Y  +349.577, Z    +0.000, E1   +27.748, E3 +36036.943}
SPL {X  -159.460, Y  +364.489, Z    +0.000, E1   +15.407, E3 +36038.238}
SPL {X  -159.962, Y  +374.520, Z    +0.000, E1    +5.534, E3 +36038.634}
SPL {X  -159.990, Y  +379.490, Z    +0.000, E1    +0.023, E3 +36038.691}
SPL {X  -159.990, Y  +381.667, Z    +0.000, E1    -4.707, E3 +36038.713}
SPL {X  -159.990, Y  +385.814, Z    +0.000, E1   -15.621, E3 +36038.817}
SPL {X  -159.990, Y  +390.948, Z    +0.000, E1   -28.850, E3 +36039.094}
SPL {X  -159.990, Y  +399.006, Z    +0.000, E1   -45.565, E3 +36039.805}
SPL {X  -159.990, Y  +410.008, Z    +0.000, E1   -58.546, E3 +36041.415}
SPL {X  -159.990, Y  +430.714, Z    +0.000, E1   -67.965, E3 +36046.221}
SPL {X  -159.990, Y  +500.758, Z    +0.000, E1   -73.927, E3 +36068.896}
SPL {X  -158.798, Y  +695.991, Z    +0.000, E1   -74.986, E3 +36156.733}
SPL {X  -156.512, Y  +709.677, Z    +0.000, E1   -74.772, E3 +36166.877}
SPL {X  -153.684, Y  +720.975, Z    +0.000, E1   -74.508, E3 +36176.164}
SPL {X  -149.353, Y  +733.863, Z    +0.000, E1   -74.100, E3 +36187.752}
SPL {X  -145.190, Y  +743.705, Z    +0.000, E1   -73.640, E3 +36197.433}
SPL {X  -141.940, Y  +750.322, Z    +0.000, E1   -73.290, E3 +36204.200}
SPL {X  -138.555, Y  +756.496, Z    +0.000, E1   -72.905, E3 +36210.765}
SPL {X  -135.025, Y  +762.319, Z    +0.000, E1   -72.483, E3 +36217.145}
SPL {X  -131.747, Y  +767.272, Z    +0.000, E1   -72.071, E3 +36222.670}
SPL {X  -128.648, Y  +771.613, Z    +0.000, E1   -71.666, E3 +36227.562}
SPL {X  -125.012, Y  +776.344, Z    +0.000, E1   -71.184, E3 +36232.873}
SPL {X  -120.782, Y  +781.422, Z    +0.000, E1   -70.584, E3 +36238.511}
SPL {X   -74.295, Y  +818.193, Z    +0.000, E1   -57.793, E3 +36348.842}
ENDSPLINE

SPLINE
SPL {X  -105.102, Y  +797.125, Z    +0.000, E1   -55.734, E3 +36528.209}
SPL {X  -126.361, Y  +774.631, Z    +0.000, E1   -54.192, E3 +36553.876}
SPL {X  -145.777, Y  +742.423, Z    +0.000, E1   -46.722, E3 +36569.217}
SPL {X  -154.920, Y  +716.458, Z    +0.000, E1   -35.175, E3 +36575.272}
SPL {X  -159.063, Y  +693.702, Z    +0.000, E1   -19.028, E3 +36578.053}
SPL {X  -159.958, Y  +679.684, Z    +0.000, E1    -5.688, E3 +36578.765}
SPL {X  -159.990, Y  +674.512, Z    +0.000, E1    -0.026, E3 +36578.830}
SPL {X  -159.990, Y  +672.767, Z    +0.000, E1    +3.705, E3 +36578.843}
SPL {X  -159.990, Y  +669.310, Z    +0.000, E1   +12.444, E3 +36578.917}
SPL {X  -159.990, Y  +665.511, Z    +0.000, E1   +22.359, E3 +36579.076}
SPL {X  -159.990, Y  +660.776, Z    +0.000, E1   +34.018, E3 +36579.383}
SPL {X  -159.990, Y  +655.863, Z    +0.000, E1   +43.768, E3 +36579.840}
SPL {X  -159.990, Y  +646.280, Z    +0.000, E1   +56.156, E3 +36581.129}
SPL {X  -159.990, Y  +625.549, Z    +0.000, E1   +67.208, E3 +36585.651}
SPL {X  -159.990, Y  +550.186, Z    +0.000, E1   +73.637, E3 +36611.057}
SPL {X  -159.878, Y  +371.520, Z    +0.000, E1   +74.559, E3 +36693.819}
SPL {X  -159.109, Y  +360.737, Z    +0.000, E1   +74.490, E3 +36700.943}
SPL {X  -156.915, Y  +346.281, Z    +0.000, E1   +74.304, E3 +36711.646}
ENDSPLINE

SPLINE
SPL {X  -159.697, Y  +367.814, Z    +0.000, E1   +71.217, E3 +36728.965}
ENDSPLINE

SPLINE
SPL {X  -157.536, Y  +349.586, Z    +0.000, E1   +71.787, E3 +36736.263}
SPL {X  -154.855, Y  +337.291, Z    +0.000, E1   +72.155, E3 +36741.017}
SPL {X  -150.925, Y  +324.412, Z    +0.000, E1   +72.419, E3 +36746.911}
SPL {X  -144.972, Y  +309.824, Z    +0.000, E1   +72.799, E3 +36752.513}
SPL {X  -139.605, Y  +299.351, Z    +0.000, E1   +73.035, E3 +36756.645}
SPL {X  -136.475, Y  +294.006, Z    +0.000, E1   +72.670, E3 +36762.430}
SPL {X  -133.214, Y  +288.895, Z    +0.000, E1   +72.272, E3 +36768.077}
SPL {X  -129.829, Y  +284.006, Z    +0.000, E1   +71.844, E3 +36773.552}
SPL {X  -126.314, Y  +279.309, Z    +0.000, E1   +71.374, E3 +36778.845}
SPL {X  -122.705, Y  +274.834, Z    +0.000, E1   +70.869, E3 +36783.856}
SPL {X  -119.804, Y  +271.463, Z    +0.000, E1   +70.429, E3 +36787.574}
SPL {X   -77.409, Y  +237.483, Z    +0.000, E1   +59.013, E3 +36881.250}
ENDSPLINE

SPLINE
SPL {X  -103.775, Y  +255.731, Z    +0.000, E1   +56.205, E3 +37077.963}
SPL {X  -141.196, Y  +302.265, Z    +0.000, E1   +49.914, E3 +37115.448}
SPL {X  -155.405, Y  +339.473, Z    +0.000, E1   +34.418, E3 +37125.149}
SPL {X  -158.399, Y  +354.990, Z    +0.000, E1   +23.559, E3 +37127.080}
SPL {X  -159.460, Y  +364.489, Z    +0.000, E1   +15.407, E3 +37127.791}
SPL {X  -159.962, Y  +374.520, Z    +0.000, E1    +5.534, E3 +37128.186}
SPL {X  -159.990, Y  +379.741, Z    +0.000, E1    -0.257, E3 +37128.245}
SPL {X  -159.990, Y  +384.604, Z    +0.000, E1   -12.124, E3 +37128.334}
SPL {X  -159.990, Y  +390.948, Z    +0.000, E1   -28.850, E3 +37128.646}
SPL {X  -159.990, Y  +399.006, Z    +0.000, E1   -45.565, E3 +37129.357}
SPL {X  -159.990, Y  +410.008, Z    +0.000, E1   -58.546, E3 +37130.968}
SPL {X  -159.990, Y  +426.664, Z    +0.000, E1   -66.963, E3 +37134.589}
SPL {X  -159.990, Y  +494.829, Z    +0.000, E1   -73.764, E3 +37156.353}
SPL {X  -158.798, Y  +695.991, Z    +0.000, E1   -74.986, E3 +37246.286}
SPL {X  -156.512, Y  +709.677, Z    +0.000, E1   -74.772, E3 +37256.429}
SPL {X  -153.684, Y  +720.975, Z    +0.000, E1   -74.508, E3 +37265.717}
SPL {X  -149.353, Y  +733.863, Z    +0.000, E1   -74.100, E3 +37277.304}
SPL {X  -145.190, Y  +743.705, Z    +0.000, E1   -73.640, E3 +37286.985}
SPL {X  -141.940, Y  +750.322, Z    +0.000, E1   -73.290, E3 +37293.752}
SPL {X  -138.555, Y  +756.496, Z    +0.000, E1   -72.905, E3 +37300.317}
SPL {X  -135.025, Y  +762.319, Z    +0.000, E1   -72.483, E3 +37306.697}
SPL {X  -131.747, Y  +767.272, Z    +0.000, E1   -72.071, E3 +37312.222}
SPL {X  -128.648, Y  +771.613, Z    +0.000, E1   -71.666, E3 +37317.114}
SPL {X  -125.012, Y  +776.344, Z    +0.000, E1   -71.184, E3 +37322.426}
SPL {X  -121.578, Y  +780.498, Z    +0.000, E1   -70.681, E3 +37327.069}
SPL {X  -119.460, Y  +782.925, Z    +0.000, E1   -70.353, E3 +37329.733}
SPL {X   -74.295, Y  +818.193, Z    +0.000, E1   -57.793, E3 +37438.394}
ENDSPLINE

SPLINE
SPL {X  -120.240, Y  +782.043, Z    +0.000, E1   -55.019, E3 +37636.890}
SPL {X  -145.777, Y  +742.423, Z    +0.000, E1   -46.722, E3 +37658.769}
SPL {X  -154.920, Y  +716.458, Z    +0.000, E1   -35.175, E3 +37664.824}
SPL {X  -159.063, Y  +693.702, Z    +0.000, E1   -19.028, E3 +37667.606}
SPL {X  -159.958, Y  +679.684, Z    +0.000, E1    -5.688, E3 +37668.318}
SPL {X  -159.990, Y  +674.512, Z    +0.000, E1    -0.026, E3 +37668.382}
SPL {X  -159.990, Y  +672.767, Z    +0.000, E1    +3.705, E3 +37668.396}
SPL {X  -159.990, Y  +669.310, Z    +0.000, E1   +12.444, E3 +37668.470}
SPL {X  -159.990, Y  +665.511, Z    +0.000, E1   +22.359, E3 +37668.628}
SPL {X  -159.990, Y  +658.432, Z    +0.000, E1   +38.720, E3 +37669.153}
SPL {X  -159.990, Y  +646.280, Z    +0.000, E1   +56.156, E3 +37670.682}
SPL {X  -159.990, Y  +625.549, Z    +0.000, E1   +67.208, E3 +37675.203}
SPL {X  -159.990, Y  +550.186, Z    +0.000, E1   +73.637, E3 +37700.609}
SPL {X  -159.493, Y  +364.902, Z    +0.000, E1   +74.541, E3 +37787.602}
SPL {X  -156.915, Y  +346.281, Z    +0.000, E1   +74.304, E3 +37801.198}
ENDSPLINE

SPLINE
SPL {X  -159.697, Y  +367.814, Z    +0.000, E1   +71.217, E3 +37818.517}
ENDSPLINE

SPLINE
SPL {X  -157.536, Y  +349.586, Z    +0.000, E1   +71.787, E3 +37825.815}
SPL {X  -154.855, Y  +337.291, Z    +0.000, E1   +72.155, E3 +37830.569}
SPL {X  -150.925, Y  +324.412, Z    +0.000, E1   +72.419, E3 +37836.463}
SPL {X  -146.819, Y  +313.931, Z    +0.000, E1   +72.621, E3 +37841.157}
SPL {X  -140.820, Y  +301.561, Z    +0.000, E1   +73.023, E3 +37845.073}
SPL {X  -136.475, Y  +294.006, Z    +0.000, E1   +72.670, E3 +37851.982}
SPL {X  -133.214, Y  +288.895, Z    +0.000, E1   +72.272, E3 +37857.630}
SPL {X  -129.829, Y  +284.006, Z    +0.000, E1   +71.844, E3 +37863.104}
SPL {X  -126.314, Y  +279.309, Z    +0.000, E1   +71.374, E3 +37868.397}
SPL {X  -122.705, Y  +274.834, Z    +0.000, E1   +70.869, E3 +37873.408}
SPL {X  -119.804, Y  +271.463, Z    +0.000, E1   +70.429, E3 +37877.127}
SPL {X   -77.409, Y  +237.483, Z    +0.000, E1   +59.013, E3 +37970.802}
ENDSPLINE

SPLINE
SPL {X  -103.775, Y  +255.731, Z    +0.000, E1   +56.205, E3 +38167.516}
SPL {X  -141.196, Y  +302.265, Z    +0.000, E1   +49.914, E3 +38205.001}
SPL {X  -155.405, Y  +339.473, Z    +0.000, E1   +34.418, E3 +38214.701}
SPL {X  -159.172, Y  +361.346, Z    +0.000, E1   +18.323, E3 +38217.126}
SPL {X  -159.962, Y  +374.520, Z    +0.000, E1    +5.534, E3 +38217.739}
SPL {X  -159.990, Y  +379.490, Z    +0.000, E1    +0.023, E3 +38217.796}
SPL {X  -159.990, Y  +381.667, Z    +0.000, E1    -4.707, E3 +38217.818}
SPL {X  -159.990, Y  +385.814, Z    +0.000, E1   -15.621, E3 +38217.922}
SPL {X  -159.990, Y  +390.948, Z    +0.000, E1   -28.850, E3 +38218.198}
SPL {X  -159.990, Y  +399.006, Z    +0.000, E1   -45.565, E3 +38218.910}
SPL {X  -159.990, Y  +410.008, Z    +0.000, E1   -58.546, E3 +38220.520}
SPL {X  -159.990, Y  +426.664, Z    +0.000, E1   -66.963, E3 +38224.141}
SPL {X  -159.990, Y  +494.829, Z    +0.000, E1   -73.764, E3 +38245.905}
SPL {X  -158.798, Y  +695.991, Z    +0.000, E1   -74.986, E3 +38335.838}
SPL {X  -156.512, Y  +709.677, Z    +0.000, E1   -74.772, E3 +38345.981}
SPL {X  -153.684, Y  +720.975, Z    +0.000, E1   -74.508, E3 +38355.269}
SPL {X  -150.879, Y  +729.719, Z    +0.000, E1   -74.224, E3 +38363.063}
SPL {X  -148.237, Y  +736.689, Z    +0.000, E1   -73.960, E3 +38369.617}
SPL {X  -145.190, Y  +743.705, Z    +0.000, E1   -73.640, E3 +38376.538}
SPL {X  -141.940, Y  +750.322, Z    +0.000, E1   -73.290, E3 +38383.304}
SPL {X  -138.555, Y  +756.496, Z    +0.000, E1   -72.905, E3 +38389.869}
SPL {X  -135.025, Y  +762.319, Z    +0.000, E1   -72.483, E3 +38396.249}
SPL {X  -131.747, Y  +767.272, Z    +0.000, E1   -72.071, E3 +38401.774}
SPL {X  -127.432, Y  +773.236, Z    +0.000, E1   -71.530, E3 +38408.459}
SPL {X  -124.036, Y  +777.554, Z    +0.000, E1   -71.026, E3 +38413.358}
SPL {X  -120.782, Y  +781.422, Z    +0.000, E1   -70.584, E3 +38417.616}
SPL {X   -74.295, Y  +818.193, Z    +0.000, E1   -57.793, E3 +38527.946}
ENDSPLINE

SPLINE
SPL {X  -105.102, Y  +797.125, Z    +0.000, E1   -55.734, E3 +38707.313}
SPL {X  -126.361, Y  +774.631, Z    +0.000, E1   -54.192, E3 +38732.981}
SPL {X  -145.777, Y  +742.423, Z    +0.000, E1   -46.722, E3 +38748.322}
SPL {X  -154.920, Y  +716.458, Z    +0.000, E1   -35.175, E3 +38754.377}
SPL {X  -159.063, Y  +693.702, Z    +0.000, E1   -19.028, E3 +38757.158}
SPL {X  -159.958, Y  +679.684, Z    +0.000, E1    -5.688, E3 +38757.870}
SPL {X  -159.990, Y  +674.512, Z    +0.000, E1    -0.026, E3 +38757.935}
SPL {X  -159.990, Y  +672.767, Z    +0.000, E1    +3.705, E3 +38757.948}
SPL {X  -159.990, Y  +669.310, Z    +0.000, E1   +12.444, E3 +38758.022}
SPL {X  -159.990, Y  +665.511, Z    +0.000, E1   +22.359, E3 +38758.180}
SPL {X  -159.990, Y  +660.776, Z    +0.000, E1   +34.018, E3 +38758.487}
SPL {X  -159.990, Y  +655.863, Z    +0.000, E1   +43.768, E3 +38758.945}
SPL {X  -159.990, Y  +646.280, Z    +0.000, E1   +56.156, E3 +38760.234}
SPL {X  -159.990, Y  +625.549, Z    +0.000, E1   +67.208, E3 +38764.756}
SPL {X  -159.990, Y  +550.186, Z    +0.000, E1   +73.637, E3 +38790.161}
SPL {X  -159.493, Y  +364.902, Z    +0.000, E1   +74.541, E3 +38877.155}
SPL {X  -156.915, Y  +346.281, Z    +0.000, E1   +74.304, E3 +38890.751}
ENDSPLINE

SPLINE
SPL {X  -159.697, Y  +367.814, Z    +0.000, E1   +71.217, E3 +38908.069}
ENDSPLINE

SPLINE
SPL {X  -157.536, Y  +349.586, Z    +0.000, E1   +71.787, E3 +38915.367}
SPL {X  -154.855, Y  +337.291, Z    +0.000, E1   +72.155, E3 +38920.121}
SPL {X  -150.925, Y  +324.412, Z    +0.000, E1   +72.419, E3 +38926.015}
SPL {X  -146.819, Y  +313.931, Z    +0.000, E1   +72.621, E3 +38930.709}
SPL {X  -140.820, Y  +301.561, Z    +0.000, E1   +73.023, E3 +38934.625}
SPL {X  -136.475, Y  +294.006, Z    +0.000, E1   +72.670, E3 +38941.534}
SPL {X  -133.214, Y  +288.895, Z    +0.000, E1   +72.272, E3 +38947.182}
SPL {X  -129.829, Y  +284.006, Z    +0.000, E1   +71.844, E3 +38952.657}
SPL {X  -126.314, Y  +279.309, Z    +0.000, E1   +71.374, E3 +38957.949}
SPL {X  -122.705, Y  +274.834, Z    +0.000, E1   +70.869, E3 +38962.960}
SPL {X  -119.804, Y  +271.463, Z    +0.000, E1   +70.429, E3 +38966.679}
SPL {X   -77.409, Y  +237.483, Z    +0.000, E1   +59.013, E3 +39060.354}
ENDSPLINE

SPLINE
SPL {X  -103.775, Y  +255.731, Z    +0.000, E1   +56.205, E3 +39257.068}
SPL {X  -141.196, Y  +302.265, Z    +0.000, E1   +49.914, E3 +39294.553}
SPL {X  -155.405, Y  +339.473, Z    +0.000, E1   +34.418, E3 +39304.253}
SPL {X  -159.172, Y  +361.346, Z    +0.000, E1   +18.323, E3 +39306.678}
SPL {X  -159.962, Y  +374.520, Z    +0.000, E1    +5.534, E3 +39307.291}
SPL {X  -159.990, Y  +379.490, Z    +0.000, E1    +0.023, E3 +39307.348}
SPL {X  -159.990, Y  +381.667, Z    +0.000, E1    -4.707, E3 +39307.370}
SPL {X  -159.990, Y  +387.434, Z    +0.000, E1   -19.600, E3 +39307.553}
SPL {X  -159.990, Y  +395.000, Z    +0.000, E1   -38.121, E3 +39308.061}
SPL {X  -159.990, Y  +406.380, Z    +0.000, E1   -55.108, E3 +39309.503}
SPL {X  -159.990, Y  +426.664, Z    +0.000, E1   -66.963, E3 +39313.693}
SPL {X  -159.990, Y  +494.829, Z    +0.000, E1   -73.764, E3 +39335.457}
SPL {X  -158.798, Y  +695.991, Z    +0.000, E1   -74.986, E3 +39425.390}
SPL {X  -156.512, Y  +709.677, Z    +0.000, E1   -74.772, E3 +39435.534}
SPL {X  -153.684, Y  +720.975, Z    +0.000, E1   -74.508, E3 +39444.821}
SPL {X  -149.353, Y  +733.863, Z    +0.000, E1   -74.100, E3 +39456.409}
SPL {X  -145.190, Y  +743.705, Z    +0.000, E1   -73.640, E3 +39466.090}
SPL {X  -141.940, Y  +750.322, Z    +0.000, E1   -73.290, E3 +39472.857}
SPL {X  -138.555, Y  +756.496, Z    +0.000, E1   -72.905, E3 +39479.422}
SPL {X  -135.025, Y  +762.319, Z    +0.000, E1   -72.483, E3 +39485.801}
SPL {X  -131.747, Y  +767.272, Z    +0.000, E1   -72.071, E3 +39491.326}
SPL {X  -127.432, Y  +773.236, Z    +0.000, E1   -71.530, E3 +39498.012}
SPL {X  -124.036, Y  +777.554, Z    +0.000, E1   -71.026, E3 +39502.910}
SPL {X  -120.782, Y  +781.422, Z    +0.000, E1   -70.584, E3 +39507.168}
SPL {X   -74.295, Y  +818.193, Z    +0.000, E1   -57.793, E3 +39617.499}
ENDSPLINE

SPLINE
SPL {X  -105.102, Y  +797.125, Z    +0.000, E1   -55.734, E3 +39796.865}
SPL {X  -126.361, Y  +774.631, Z    +0.000, E1   -54.192, E3 +39822.533}
SPL {X  -145.777, Y  +742.423, Z    +0.000, E1   -46.722, E3 +39837.874}
SPL {X  -154.920, Y  +716.458, Z    +0.000, E1   -35.175, E3 +39843.929}
SPL {X  -159.063, Y  +693.702, Z    +0.000, E1   -19.028, E3 +39846.710}
SPL {X  -159.958, Y  +679.684, Z    +0.000, E1    -5.688, E3 +39847.422}
SPL {X  -159.990, Y  +674.512, Z    +0.000, E1    -0.026, E3 +39847.487}
SPL {X  -159.990, Y  +672.767, Z    +0.000, E1    +3.705, E3 +39847.500}
SPL {X  -159.990, Y  +669.310, Z    +0.000, E1   +12.444, E3 +39847.574}
SPL {X  -159.990, Y  +665.511, Z    +0.000, E1   +22.359, E3 +39847.733}
SPL {X  -159.990, Y  +660.776, Z    +0.000, E1   +34.018, E3 +39848.039}
SPL {X  -159.990, Y  +655.863, Z    +0.000, E1   +43.768, E3 +39848.497}
SPL {X  -159.990, Y  +646.280, Z    +0.000, E1   +56.156, E3 +39849.786}
SPL {X  -159.990, Y  +625.549, Z    +0.000, E1   +67.208, E3 +39854.308}
SPL {X  -159.990, Y  +550.186, Z    +0.000, E1   +73.637, E3 +39879.714}
SPL {X  -159.493, Y  +364.902, Z    +0.000, E1   +74.541, E3 +39966.707}
SPL {X  -156.915, Y  +346.281, Z    +0.000, E1   +74.304, E3 +39980.303}
ENDSPLINE

SPLINE
SPL {X  -159.697, Y  +367.814, Z    +0.000, E1   +71.217, E3 +39997.621}
ENDSPLINE

SPLINE
SPL {X  -157.536, Y  +349.586, Z    +0.000, E1   +71.787, E3 +40004.919}
SPL {X  -154.855, Y  +337.291, Z    +0.000, E1   +72.155, E3 +40009.673}
SPL {X  -150.925, Y  +324.412, Z    +0.000, E1   +72.419, E3 +40015.568}
SPL {X  -146.819, Y  +313.931, Z    +0.000, E1   +72.621, E3 +40020.261}
SPL {X  -140.820, Y  +301.561, Z    +0.000, E1   +73.023, E3 +40024.177}
SPL {X  -136.475, Y  +294.006, Z    +0.000, E1   +72.670, E3 +40031.086}
SPL {X  -133.214, Y  +288.895, Z    +0.000, E1   +72.272, E3 +40036.734}
SPL {X  -129.829, Y  +284.006, Z    +0.000, E1   +71.844, E3 +40042.209}
SPL {X  -126.314, Y  +279.309, Z    +0.000, E1   +71.374, E3 +40047.501}
SPL {X  -122.705, Y  +274.834, Z    +0.000, E1   +70.869, E3 +40052.512}
SPL {X  -119.804, Y  +271.463, Z    +0.000, E1   +70.429, E3 +40056.231}
SPL {X   -77.409, Y  +237.483, Z    +0.000, E1   +59.013, E3 +40149.907}
ENDSPLINE

SPLINE
SPL {X  -103.775, Y  +255.731, Z    +0.000, E1   +56.205, E3 +40346.620}
SPL {X  -141.196, Y  +302.265, Z    +0.000, E1   +49.914, E3 +40384.105}
SPL {X  -155.405, Y  +339.473, Z    +0.000, E1   +34.418, E3 +40393.805}
SPL {X  -159.172, Y  +361.346, Z    +0.000, E1   +18.323, E3 +40396.230}
SPL {X  -159.962, Y  +374.520, Z    +0.000, E1    +5.534, E3 +40396.843}
SPL {X  -159.990, Y  +379.490, Z    +0.000, E1    +0.023, E3 +40396.900}
SPL {X  -159.990, Y  +381.667, Z    +0.000, E1    -4.707, E3 +40396.922}
SPL {X  -159.990, Y  +387.434, Z    +0.000, E1   -19.600, E3 +40397.105}
SPL {X  -159.990, Y  +395.000, Z    +0.000, E1   -38.121, E3 +40397.614}
SPL {X  -159.990, Y  +406.380, Z    +0.000, E1   -55.108, E3 +40399.055}
SPL {X  -159.990, Y  +426.664, Z    +0.000, E1   -66.963, E3 +40403.246}
SPL {X  -159.990, Y  +494.829, Z    +0.000, E1   -73.764, E3 +40425.010}
SPL {X  -158.798, Y  +695.991, Z    +0.000, E1   -74.986, E3 +40514.942}
SPL {X  -156.512, Y  +709.677, Z    +0.000, E1   -74.772, E3 +40525.086}
SPL {X  -153.684, Y  +720.975, Z    +0.000, E1   -74.508, E3 +40534.373}
SPL {X  -149.353, Y  +733.863, Z    +0.000, E1   -74.100, E3 +40545.961}
SPL {X  -145.190, Y  +743.705, Z    +0.000, E1   -73.640, E3 +40555.642}
SPL {X  -141.940, Y  +750.322, Z    +0.000, E1   -73.290, E3 +40562.409}
SPL {X  -138.555, Y  +756.496, Z    +0.000, E1   -72.905, E3 +40568.974}
SPL {X  -135.025, Y  +762.319, Z    +0.000, E1   -72.483, E3 +40575.354}
SPL {X  -131.747, Y  +767.272, Z    +0.000, E1   -72.071, E3 +40580.879}
SPL {X  -127.432, Y  +773.236, Z    +0.000, E1   -71.530, E3 +40587.564}
SPL {X  -124.036, Y  +777.554, Z    +0.000, E1   -71.026, E3 +40592.462}
SPL {X  -120.782, Y  +781.422, Z    +0.000, E1   -70.584, E3 +40596.720}
SPL {X   -74.295, Y  +818.193, Z    +0.000, E1   -57.793, E3 +40707.051}
ENDSPLINE

SPLINE
SPL {X  -105.102, Y  +797.125, Z    +0.000, E1   -55.734, E3 +40886.418}
SPL {X  -126.361, Y  +774.631, Z    +0.000, E1   -54.192, E3 +40912.085}
SPL {X  -145.777, Y  +742.423, Z    +0.000, E1   -46.722, E3 +40927.426}
SPL {X  -154.920, Y  +716.458, Z    +0.000, E1   -35.175, E3 +40933.481}
SPL {X  -158.252, Y  +700.019, Z    +0.000, E1   -24.087, E3 +40935.733}
SPL {X  -159.434, Y  +689.826, Z    +0.000, E1   -15.506, E3 +40936.551}
SPL {X  -159.958, Y  +679.684, Z    +0.000, E1    -5.688, E3 +40936.974}
SPL {X  -159.990, Y  +674.512, Z    +0.000, E1    -0.026, E3 +40937.039}
SPL {X  -159.990, Y  +672.767, Z    +0.000, E1    +3.705, E3 +40937.052}
SPL {X  -159.990, Y  +669.310, Z    +0.000, E1   +12.444, E3 +40937.126}
SPL {X  -159.990, Y  +665.511, Z    +0.000, E1   +22.359, E3 +40937.285}
SPL {X  -159.990, Y  +660.776, Z    +0.000, E1   +34.018, E3 +40937.592}
SPL {X  -159.990, Y  +655.863, Z    +0.000, E1   +43.768, E3 +40938.049}
SPL {X  -159.990, Y  +646.280, Z    +0.000, E1   +56.156, E3 +40939.338}
SPL {X  -159.990, Y  +625.549, Z    +0.000, E1   +67.208, E3 +40943.860}
SPL {X  -159.990, Y  +550.186, Z    +0.000, E1   +73.637, E3 +40969.266}
SPL {X  -159.878, Y  +371.520, Z    +0.000, E1   +74.559, E3 +41052.028}
SPL {X  -159.109, Y  +360.737, Z    +0.000, E1   +74.490, E3 +41059.152}
SPL {X  -156.915, Y  +346.281, Z    +0.000, E1   +74.304, E3 +41069.855}
ENDSPLINE

SPLINE
SPL {X  -159.697, Y  +367.814, Z    +0.000, E1   +71.217, E3 +41087.174}
ENDSPLINE

SPLINE
SPL {X  -156.028, Y  +342.114, Z    +0.000, E1   +72.020, E3 +41097.327}
SPL {X  -150.925, Y  +324.412, Z    +0.000, E1   +72.419, E3 +41105.120}
SPL {X  -146.819, Y  +313.931, Z    +0.000, E1   +72.621, E3 +41109.813}
SPL {X  -140.820, Y  +301.561, Z    +0.000, E1   +73.023, E3 +41113.730}
SPL {X  -136.475, Y  +294.006, Z    +0.000, E1   +72.670, E3 +41120.639}
SPL {X  -133.214, Y  +288.895, Z    +0.000, E1   +72.272, E3 +41126.286}
SPL {X  -129.829, Y  +284.006, Z    +0.000, E1   +71.844, E3 +41131.761}
SPL {X  -125.428, Y  +278.179, Z    +0.000, E1   +71.273, E3 +41138.299}
SPL {X  -120.729, Y  +272.518, Z    +0.000, E1   +70.593, E3 +41144.608}
SPL {X   -77.409, Y  +237.483, Z    +0.000, E1   +59.013, E3 +41239.459}
ENDSPLINE

SPLINE
SPL {X  -103.775, Y  +255.731, Z    +0.000, E1   +56.205, E3 +41436.172}
SPL {X  -141.196, Y  +302.265, Z    +0.000, E1   +49.914, E3 +41473.657}
SPL {X  -155.405, Y  +339.473, Z    +0.000, E1   +34.418, E3 +41483.358}
SPL {X  -159.172, Y  +361.346, Z    +0.000, E1   +18.323, E3 +41485.782}
SPL {X  -159.962, Y  +374.520, Z    +0.000, E1    +5.534, E3 +41486.395}
SPL {X  -159.990, Y  +379.490, Z    +0.000, E1    +0.023, E3 +41486.453}
SPL {X  -159.990, Y  +381.667, Z    +0.000, E1    -4.707, E3 +41486.475}
SPL {X  -159.990, Y  +385.814, Z    +0.000, E1   -15.621, E3 +41486.578}
SPL {X  -159.990, Y  +390.948, Z    +0.000, E1   -28.850, E3 +41486.855}
SPL {X  -159.990, Y  +399.006, Z    +0.000, E1   -45.565, E3 +41487.566}
SPL {X  -159.990, Y  +410.008, Z    +0.000, E1   -58.546, E3 +41489.177}
SPL {X  -159.990, Y  +426.664, Z    +0.000, E1   -66.963, E3 +41492.798}
SPL {X  -159.990, Y  +494.829, Z    +0.000, E1   -73.764, E3 +41514.562}
SPL {X  -158.798, Y  +695.991, Z    +0.000, E1   -74.986, E3 +41604.495}
SPL {X  -156.512, Y  +709.677, Z    +0.000, E1   -74.772, E3 +41614.638}
SPL {X  -153.684, Y  +720.975, Z    +0.000, E1   -74.508, E3 +41623.926}
SPL {X  -149.353, Y  +733.863, Z    +0.000, E1   -74.100, E3 +41635.513}
SPL {X  -145.190, Y  +743.705, Z    +0.000, E1   -73.640, E3 +41645.194}
SPL {X  -141.940, Y  +750.322, Z    +0.000, E1   -73.290, E3 +41651.961}
SPL {X  -138.555, Y  +756.496, Z    +0.000, E1   -72.905, E3 +41658.526}
SPL {X  -135.025, Y  +762.319, Z    +0.000, E1   -72.483, E3 +41664.906}
SPL {X  -131.747, Y  +767.272, Z    +0.000, E1   -72.071, E3 +41670.431}
SPL {X  -127.432, Y  +773.236, Z    +0.000, E1   -71.530, E3 +41677.116}
SPL {X  -124.036, Y  +777.554, Z    +0.000, E1   -71.026, E3 +41682.015}
SPL {X  -120.782, Y  +781.422, Z    +0.000, E1   -70.584, E3 +41686.272}
SPL {X   -74.295, Y  +818.193, Z    +0.000, E1   -57.793, E3 +41796.603}
ENDSPLINE

SPLINE
SPL {X  -120.240, Y  +782.043, Z    +0.000, E1   -55.019, E3 +41995.099}
SPL {X  -145.777, Y  +742.423, Z    +0.000, E1   -46.722, E3 +42016.978}
SPL {X  -154.920, Y  +716.458, Z    +0.000, E1   -35.175, E3 +42023.033}
SPL {X  -158.252, Y  +700.019, Z    +0.000, E1   -24.087, E3 +42025.285}
SPL {X  -159.434, Y  +689.826, Z    +0.000, E1   -15.506, E3 +42026.103}
SPL {X  -159.958, Y  +679.684, Z    +0.000, E1    -5.688, E3 +42026.527}
SPL {X  -159.990, Y  +674.512, Z    +0.000, E1    -0.026, E3 +42026.591}
SPL {X  -159.990, Y  +672.767, Z    +0.000, E1    +3.705, E3 +42026.605}
SPL {X  -159.990, Y  +669.310, Z    +0.000, E1   +12.444, E3 +42026.678}
SPL {X  -159.990, Y  +665.511, Z    +0.000, E1   +22.359, E3 +42026.837}
SPL {X  -159.990, Y  +658.432, Z    +0.000, E1   +38.720, E3 +42027.362}
SPL {X  -159.990, Y  +646.280, Z    +0.000, E1   +56.156, E3 +42028.891}
SPL {X  -159.990, Y  +625.549, Z    +0.000, E1   +67.208, E3 +42033.412}
SPL {X  -159.990, Y  +550.186, Z    +0.000, E1   +73.637, E3 +42058.818}
SPL {X  -159.493, Y  +364.902, Z    +0.000, E1   +74.541, E3 +42145.811}
SPL {X  -156.915, Y  +346.281, Z    +0.000, E1   +74.304, E3 +42159.407}
ENDSPLINE

SPLINE
SPL {X  -159.697, Y  +367.814, Z    +0.000, E1   +71.217, E3 +42176.726}
ENDSPLINE

SPLINE
SPL {X  -156.028, Y  +342.114, Z    +0.000, E1   +72.020, E3 +42186.879}
SPL {X  -150.925, Y  +324.412, Z    +0.000, E1   +72.419, E3 +42194.672}
SPL {X  -146.819, Y  +313.931, Z    +0.000, E1   +72.621, E3 +42199.365}
SPL {X  -140.820, Y  +301.561, Z    +0.000, E1   +73.023, E3 +42203.282}
SPL {X  -136.475, Y  +294.006, Z    +0.000, E1   +72.670, E3 +42210.191}
SPL {X  -133.214, Y  +288.895, Z    +0.000, E1   +72.272, E3 +42215.839}
SPL {X  -129.829, Y  +284.006, Z    +0.000, E1   +71.844, E3 +42221.313}
SPL {X  -126.314, Y  +279.309, Z    +0.000, E1   +71.374, E3 +42226.606}
SPL {X  -122.705, Y  +274.834, Z    +0.000, E1   +70.869, E3 +42231.617}
SPL {X  -119.804, Y  +271.463, Z    +0.000, E1   +70.429, E3 +42235.336}
SPL {X   -77.409, Y  +237.483, Z    +0.000, E1   +59.013, E3 +42329.011}
ENDSPLINE

SPLINE
SPL {X  -103.775, Y  +255.731, Z    +0.000, E1   +56.205, E3 +42525.724}
SPL {X  -141.196, Y  +302.265, Z    +0.000, E1   +49.914, E3 +42563.210}
SPL {X  -155.405, Y  +339.473, Z    +0.000, E1   +34.418, E3 +42572.910}
SPL {X  -159.172, Y  +361.346, Z    +0.000, E1   +18.323, E3 +42575.335}
SPL {X  -159.962, Y  +374.520, Z    +0.000, E1    +5.534, E3 +42575.948}
SPL {X  -159.990, Y  +379.741, Z    +0.000, E1    -0.257, E3 +42576.006}
SPL {X  -159.990, Y  +384.604, Z    +0.000, E1   -12.124, E3 +42576.095}
SPL {X  -159.990, Y  +390.948, Z    +0.000, E1   -28.850, E3 +42576.407}
SPL {X  -159.990, Y  +399.006, Z    +0.000, E1   -45.565, E3 +42577.119}
SPL {X  -159.990, Y  +410.008, Z    +0.000, E1   -58.546, E3 +42578.729}
SPL {X  -159.990, Y  +426.664, Z    +0.000, E1   -66.963, E3 +42582.350}
SPL {X  -159.990, Y  +494.829, Z    +0.000, E1   -73.764, E3 +42604.114}
SPL {X  -158.798, Y  +695.991, Z    +0.000, E1   -74.986, E3 +42694.047}
SPL {X  -156.512, Y  +709.677, Z    +0.000, E1   -74.772, E3 +42704.190}
SPL {X  -153.684, Y  +720.975, Z    +0.000, E1   -74.508, E3 +42713.478}
SPL {X  -149.353, Y  +733.863, Z    +0.000, E1   -74.100, E3 +42725.066}
SPL {X  -145.190, Y  +743.705, Z    +0.000, E1   -73.640, E3 +42734.747}
SPL {X  -141.940, Y  +750.322, Z    +0.000, E1   -73.290, E3 +42741.513}
SPL {X  -138.555, Y  +756.496, Z    +0.000, E1   -72.905, E3 +42748.078}
SPL {X  -135.025, Y  +762.319, Z    +0.000, E1   -72.483, E3 +42754.458}
SPL {X  -131.747, Y  +767.272, Z    +0.000, E1   -72.071, E3 +42759.983}
SPL {X  -128.648, Y  +771.613, Z    +0.000, E1   -71.666, E3 +42764.875}
SPL {X  -125.012, Y  +776.344, Z    +0.000, E1   -71.184, E3 +42770.187}
SPL {X  -120.782, Y  +781.422, Z    +0.000, E1   -70.584, E3 +42775.825}
SPL {X   -74.295, Y  +818.193, Z    +0.000, E1   -57.793, E3 +42886.155}
ENDSPLINE

SPLINE
SPL {X  -120.240, Y  +782.043, Z    +0.000, E1   -55.019, E3 +43084.651}
SPL {X  -145.777, Y  +742.423, Z    +0.000, E1   -46.722, E3 +43106.531}
SPL {X  -154.920, Y  +716.458, Z    +0.000, E1   -35.175, E3 +43112.586}
SPL {X  -159.063, Y  +693.702, Z    +0.000, E1   -19.028, E3 +43115.367}
SPL {X  -159.958, Y  +679.684, Z    +0.000, E1    -5.688, E3 +43116.079}
SPL {X  -159.990, Y  +674.512, Z    +0.000, E1    -0.026, E3 +43116.143}
SPL {X  -159.990, Y  +672.767, Z    +0.000, E1    +3.705, E3 +43116.157}
SPL {X  -159.990, Y  +669.310, Z    +0.000, E1   +12.444, E3 +43116.231}
SPL {X  -159.990, Y  +665.511, Z    +0.000, E1   +22.359, E3 +43116.389}
SPL {X  -159.990, Y  +658.432, Z    +0.000, E1   +38.720, E3 +43116.914}
SPL {X  -159.990, Y  +646.280, Z    +0.000, E1   +56.156, E3 +43118.443}
SPL {X  -159.990, Y  +625.549, Z    +0.000, E1   +67.208, E3 +43122.965}
SPL {X  -159.990, Y  +550.186, Z    +0.000, E1   +73.637, E3 +43148.370}
SPL {X  -159.493, Y  +364.902, Z    +0.000, E1   +74.541, E3 +43235.364}
SPL {X  -156.915, Y  +346.281, Z    +0.000, E1   +74.304, E3 +43248.960}
ENDSPLINE

SPLINE
SPL {X  -159.697, Y  +367.814, Z    +0.000, E1   +71.217, E3 +43266.278}
ENDSPLINE

SPLINE
SPL {X  -157.536, Y  +349.586, Z    +0.000, E1   +71.787, E3 +43273.576}
SPL {X  -154.855, Y  +337.291, Z    +0.000, E1   +72.155, E3 +43278.330}
SPL {X  -150.925, Y  +324.412, Z    +0.000, E1   +72.419, E3 +43284.224}
SPL {X  -146.819, Y  +313.931, Z    +0.000, E1   +72.621, E3 +43288.918}
SPL {X  -140.820, Y  +301.561, Z    +0.000, E1   +73.023, E3 +43292.834}
SPL {X  -136.475, Y  +294.006, Z    +0.000, E1   +72.670, E3 +43299.743}
SPL {X  -133.214, Y  +288.895, Z    +0.000, E1   +72.272, E3 +43305.391}
SPL {X  -129.829, Y  +284.006, Z    +0.000, E1   +71.844, E3 +43310.866}
SPL {X  -126.314, Y  +279.309, Z    +0.000, E1   +71.374, E3 +43316.158}
SPL {X  -122.705, Y  +274.834, Z    +0.000, E1   +70.869, E3 +43321.169}
SPL {X  -119.804, Y  +271.463, Z    +0.000, E1   +70.429, E3 +43324.888}
SPL {X   -77.409, Y  +237.483, Z    +0.000, E1   +59.013, E3 +43418.563}
ENDSPLINE

SPLINE
SPL {X  -103.775, Y  +255.731, Z    +0.000, E1   +56.205, E3 +43615.277}
SPL {X  -141.196, Y  +302.265, Z    +0.000, E1   +49.914, E3 +43652.762}
SPL {X  -155.405, Y  +339.473, Z    +0.000, E1   +34.418, E3 +43662.462}
SPL {X  -159.172, Y  +361.346, Z    +0.000, E1   +18.323, E3 +43664.887}
SPL {X  -159.962, Y  +374.520, Z    +0.000, E1    +5.534, E3 +43665.500}
SPL {X  -159.990, Y  +379.490, Z    +0.000, E1    +0.023, E3 +43665.557}
SPL {X  -159.990, Y  +381.667, Z    +0.000, E1    -4.707, E3 +43665.579}
SPL {X  -159.990, Y  +385.814, Z    +0.000, E1   -15.621, E3 +43665.683}
SPL {X  -159.990, Y  +390.948, Z    +0.000, E1   -28.850, E3 +43665.959}
SPL {X  -159.990, Y  +399.006, Z    +0.000, E1   -45.565, E3 +43666.671}
SPL {X  -159.990, Y  +410.008, Z    +0.000, E1   -58.546, E3 +43668.281}
SPL {X  -159.990, Y  +426.664, Z    +0.000, E1   -66.963, E3 +43671.902}
SPL {X  -159.990, Y  +494.829, Z    +0.000, E1   -73.764, E3 +43693.666}
SPL {X  -158.798, Y  +695.991, Z    +0.000, E1   -74.986, E3 +43783.599}
SPL {X  -156.512, Y  +709.677, Z    +0.000, E1   -74.772, E3 +43793.743}
SPL {X  -153.684, Y  +720.975, Z    +0.000, E1   -74.508, E3 +43803.030}
SPL {X  -150.879, Y  +729.719, Z    +0.000, E1   -74.224, E3 +43810.824}
SPL {X  -148.237, Y  +736.689, Z    +0.000, E1   -73.960, E3 +43817.378}
SPL {X  -145.190, Y  +743.705, Z    +0.000, E1   -73.640, E3 +43824.299}
SPL {X  -141.940, Y  +750.322, Z    +0.000, E1   -73.290, E3 +43831.066}
SPL {X  -138.555, Y  +756.496, Z    +0.000, E1   -72.905, E3 +43837.631}
SPL {X  -135.025, Y  +762.319, Z    +0.000, E1   -72.483, E3 +43844.010}
SPL {X  -131.747, Y  +767.272, Z    +0.000, E1   -72.071, E3 +43849.535}
SPL {X  -128.648, Y  +771.613, Z    +0.000, E1   -71.666, E3 +43854.428}
SPL {X  -125.012, Y  +776.344, Z    +0.000, E1   -71.184, E3 +43859.739}
SPL {X  -120.782, Y  +781.422, Z    +0.000, E1   -70.584, E3 +43865.377}
SPL {X   -74.295, Y  +818.193, Z    +0.000, E1   -57.793, E3 +43975.708}
ENDSPLINE

SPLINE
SPL {X  -120.240, Y  +782.043, Z    +0.000, E1   -55.019, E3 +44174.203}
SPL {X  -145.777, Y  +742.423, Z    +0.000, E1   -46.722, E3 +44196.083}
SPL {X  -154.920, Y  +716.458, Z    +0.000, E1   -35.175, E3 +44202.138}
SPL {X  -159.063, Y  +693.702, Z    +0.000, E1   -19.028, E3 +44204.919}
SPL {X  -159.958, Y  +679.684, Z    +0.000, E1    -5.688, E3 +44205.631}
SPL {X  -159.990, Y  +674.512, Z    +0.000, E1    -0.026, E3 +44205.696}
SPL {X  -159.990, Y  +672.767, Z    +0.000, E1    +3.705, E3 +44205.709}
SPL {X  -159.990, Y  +669.310, Z    +0.000, E1   +12.444, E3 +44205.783}
SPL {X  -159.990, Y  +665.511, Z    +0.000, E1   +22.359, E3 +44205.942}
SPL {X  -159.990, Y  +658.432, Z    +0.000, E1   +38.720, E3 +44206.467}
SPL {X  -159.990, Y  +646.280, Z    +0.000, E1   +56.156, E3 +44207.995}
SPL {X  -159.990, Y  +625.549, Z    +0.000, E1   +67.208, E3 +44212.517}
SPL {X  -159.990, Y  +550.186, Z    +0.000, E1   +73.637, E3 +44237.923}
SPL {X  -159.493, Y  +364.902, Z    +0.000, E1   +74.541, E3 +44324.916}
SPL {X  -156.915, Y  +346.281, Z    +0.000, E1   +74.304, E3 +44338.512}
ENDSPLINE

SPLINE
SPL {X  -159.697, Y  +367.814, Z    +0.000, E1   +71.217, E3 +44355.830}
ENDSPLINE

SPLINE
SPL {X  -157.536, Y  +349.586, Z    +0.000, E1   +71.787, E3 +44363.128}
SPL {X  -154.855, Y  +337.291, Z    +0.000, E1   +72.155, E3 +44367.882}
SPL {X  -150.925, Y  +324.412, Z    +0.000, E1   +72.419, E3 +44373.777}
SPL {X  -146.819, Y  +313.931, Z    +0.000, E1   +72.621, E3 +44378.470}
SPL {X  -140.820, Y  +301.561, Z    +0.000, E1   +73.023, E3 +44382.386}
SPL {X  -136.475, Y  +294.006, Z    +0.000, E1   +72.670, E3 +44389.295}
SPL {X  -133.214, Y  +288.895, Z    +0.000, E1   +72.272, E3 +44394.943}
SPL {X  -129.829, Y  +284.006, Z    +0.000, E1   +71.844, E3 +44400.418}
SPL {X  -126.314, Y  +279.309, Z    +0.000, E1   +71.374, E3 +44405.710}
SPL {X  -122.705, Y  +274.834, Z    +0.000, E1   +70.869, E3 +44410.721}
SPL {X  -119.804, Y  +271.463, Z    +0.000, E1   +70.429, E3 +44414.440}
SPL {X   -77.409, Y  +237.483, Z    +0.000, E1   +59.013, E3 +44508.116}
ENDSPLINE

SPLINE
SPL {X  -103.775, Y  +255.731, Z    +0.000, E1   +56.205, E3 +44704.829}
SPL {X  -141.196, Y  +302.265, Z    +0.000, E1   +49.914, E3 +44742.314}
SPL {X  -155.405, Y  +339.473, Z    +0.000, E1   +34.418, E3 +44752.014}
SPL {X  -159.172, Y  +361.346, Z    +0.000, E1   +18.323, E3 +44754.439}
SPL {X  -159.962, Y  +374.520, Z    +0.000, E1    +5.534, E3 +44755.052}
SPL {X  -159.990, Y  +379.490, Z    +0.000, E1    +0.023, E3 +44755.109}
SPL {X  -159.990, Y  +381.667, Z    +0.000, E1    -4.707, E3 +44755.131}
SPL {X  -159.990, Y  +385.814, Z    +0.000, E1   -15.621, E3 +44755.235}
SPL {X  -159.990, Y  +390.948, Z    +0.000, E1   -28.850, E3 +44755.511}
SPL {X  -159.990, Y  +399.006, Z    +0.000, E1   -45.565, E3 +44756.223}
SPL {X  -159.990, Y  +410.008, Z    +0.000, E1   -58.546, E3 +44757.833}
SPL {X  -159.990, Y  +426.664, Z    +0.000, E1   -66.963, E3 +44761.455}
SPL {X  -159.990, Y  +494.829, Z    +0.000, E1   -73.764, E3 +44783.219}
SPL {X  -158.798, Y  +695.991, Z    +0.000, E1   -74.986, E3 +44873.151}
SPL {X  -156.512, Y  +709.677, Z    +0.000, E1   -74.772, E3 +44883.295}
SPL {X  -153.684, Y  +720.975, Z    +0.000, E1   -74.508, E3 +44892.582}
SPL {X  -149.353, Y  +733.863, Z    +0.000, E1   -74.100, E3 +44904.170}
SPL {X  -145.190, Y  +743.705, Z    +0.000, E1   -73.640, E3 +44913.851}
SPL {X  -141.940, Y  +750.322, Z    +0.000, E1   -73.290, E3 +44920.618}
SPL {X  -138.555, Y  +756.496, Z    +0.000, E1   -72.905, E3 +44927.183}
SPL {X  -135.025, Y  +762.319, Z    +0.000, E1   -72.483, E3 +44933.562}
SPL {X  -131.747, Y  +767.272, Z    +0.000, E1   -72.071, E3 +44939.087}
SPL {X  -127.432, Y  +773.236, Z    +0.000, E1   -71.530, E3 +44945.773}
SPL {X  -124.036, Y  +777.554, Z    +0.000, E1   -71.026, E3 +44950.671}
SPL {X  -120.782, Y  +781.422, Z    +0.000, E1   -70.584, E3 +44954.929}
SPL {X   -74.295, Y  +818.193, Z    +0.000, E1   -57.793, E3 +45065.260}
ENDSPLINE

SPLINE
SPL {X  -105.102, Y  +797.125, Z    +0.000, E1   -55.734, E3 +45244.627}
SPL {X  -126.361, Y  +774.631, Z    +0.000, E1   -54.192, E3 +45270.294}
SPL {X  -145.777, Y  +742.423, Z    +0.000, E1   -46.722, E3 +45285.635}
SPL {X  -154.920, Y  +716.458, Z    +0.000, E1   -35.175, E3 +45291.690}
SPL {X  -159.063, Y  +693.702, Z    +0.000, E1   -19.028, E3 +45294.471}
SPL {X  -159.958, Y  +679.684, Z    +0.000, E1    -5.688, E3 +45295.183}
SPL {X  -159.990, Y  +674.512, Z    +0.000, E1    -0.026, E3 +45295.248}
SPL {X  -159.990, Y  +672.767, Z    +0.000, E1    +3.705, E3 +45295.261}
SPL {X  -159.990, Y  +669.310, Z    +0.000, E1   +12.444, E3 +45295.335}
SPL {X  -159.990, Y  +665.511, Z    +0.000, E1   +22.359, E3 +45295.494}
SPL {X  -159.990, Y  +658.432, Z    +0.000, E1   +38.720, E3 +45296.019}
SPL {X  -159.990, Y  +646.280, Z    +0.000, E1   +56.156, E3 +45297.547}
SPL {X  -159.990, Y  +625.549, Z    +0.000, E1   +67.208, E3 +45302.069}
SPL {X  -159.990, Y  +550.186, Z    +0.000, E1   +73.637, E3 +45327.475}
SPL {X  -159.878, Y  +371.520, Z    +0.000, E1   +74.559, E3 +45410.237}
SPL {X  -159.109, Y  +360.737, Z    +0.000, E1   +74.490, E3 +45417.361}
SPL {X  -156.915, Y  +346.281, Z    +0.000, E1   +74.304, E3 +45428.064}
ENDSPLINE

SPLINE
SPL {X  -159.697, Y  +367.814, Z    +0.000, E1   +71.217, E3 +45445.383}
ENDSPLINE

SPLINE
SPL {X  -156.028, Y  +342.114, Z    +0.000, E1   +72.020, E3 +45455.536}
SPL {X  -150.925, Y  +324.412, Z    +0.000, E1   +72.419, E3 +45463.329}
SPL {X  -144.972, Y  +309.824, Z    +0.000, E1   +72.799, E3 +45468.931}
SPL {X  -139.605, Y  +299.351, Z    +0.000, E1   +73.035, E3 +45473.063}
SPL {X  -136.475, Y  +294.006, Z    +0.000, E1   +72.670, E3 +45478.847}
SPL {X  -133.214, Y  +288.895, Z    +0.000, E1   +72.272, E3 +45484.495}
SPL {X  -129.829, Y  +284.006, Z    +0.000, E1   +71.844, E3 +45489.970}
SPL {X  -125.428, Y  +278.179, Z    +0.000, E1   +71.273, E3 +45496.508}
SPL {X  -120.729, Y  +272.518, Z    +0.000, E1   +70.593, E3 +45502.817}
SPL {X   -77.409, Y  +237.483, Z    +0.000, E1   +59.013, E3 +45597.668}
ENDSPLINE

SPLINE
SPL {X  -103.775, Y  +255.731, Z    +0.000, E1   +56.205, E3 +45794.381}
SPL {X  -141.196, Y  +302.265, Z    +0.000, E1   +49.914, E3 +45831.866}
SPL {X  -155.405, Y  +339.473, Z    +0.000, E1   +34.418, E3 +45841.567}
SPL {X  -159.172, Y  +361.346, Z    +0.000, E1   +18.323, E3 +45843.991}
SPL {X  -159.962, Y  +374.520, Z    +0.000, E1    +5.534, E3 +45844.604}
SPL {X  -159.990, Y  +379.490, Z    +0.000, E1    +0.023, E3 +45844.662}
SPL {X  -159.990, Y  +381.667, Z    +0.000, E1    -4.707, E3 +45844.684}
SPL {X  -159.990, Y  +385.814, Z    +0.000, E1   -15.621, E3 +45844.787}
SPL {X  -159.990, Y  +390.948, Z    +0.000, E1   -28.850, E3 +45845.064}
SPL {X  -159.990, Y  +399.006, Z    +0.000, E1   -45.565, E3 +45845.775}
SPL {X  -159.990, Y  +410.008, Z    +0.000, E1   -58.546, E3 +45847.386}
SPL {X  -159.990, Y  +426.664, Z    +0.000, E1   -66.963, E3 +45851.007}
SPL {X  -159.990, Y  +494.829, Z    +0.000, E1   -73.764, E3 +45872.771}
SPL {X  -158.798, Y  +695.991, Z    +0.000, E1   -74.986, E3 +45962.704}
SPL {X  -156.512, Y  +709.677, Z    +0.000, E1   -74.772, E3 +45972.847}
SPL {X  -153.684, Y  +720.975, Z    +0.000, E1   -74.508, E3 +45982.134}
SPL {X  -149.353, Y  +733.863, Z    +0.000, E1   -74.100, E3 +45993.722}
SPL {X  -145.190, Y  +743.705, Z    +0.000, E1   -73.640, E3 +46003.403}
SPL {X  -141.940, Y  +750.322, Z    +0.000, E1   -73.290, E3 +46010.170}
SPL {X  -138.555, Y  +756.496, Z    +0.000, E1   -72.905, E3 +46016.735}
SPL {X  -135.025, Y  +762.319, Z    +0.000, E1   -72.483, E3 +46023.115}
SPL {X  -131.747, Y  +767.272, Z    +0.000, E1   -72.071, E3 +46028.640}
SPL {X  -127.432, Y  +773.236, Z    +0.000, E1   -71.530, E3 +46035.325}
SPL {X  -124.036, Y  +777.554, Z    +0.000, E1   -71.026, E3 +46040.224}
SPL {X  -120.782, Y  +781.422, Z    +0.000, E1   -70.584, E3 +46044.481}
SPL {X   -74.295, Y  +818.193, Z    +0.000, E1   -57.793, E3 +46154.812}
ENDSPLINE

SPLINE
SPL {X  -105.102, Y  +797.125, Z    +0.000, E1   -55.734, E3 +46334.179}
SPL {X  -126.361, Y  +774.631, Z    +0.000, E1   -54.192, E3 +46359.846}
SPL {X  -145.777, Y  +742.423, Z    +0.000, E1   -46.722, E3 +46375.187}
SPL {X  -154.920, Y  +716.458, Z    +0.000, E1   -35.175, E3 +46381.242}
SPL {X  -159.063, Y  +693.702, Z    +0.000, E1   -19.028, E3 +46384.024}
SPL {X  -159.958, Y  +679.684, Z    +0.000, E1    -5.688, E3 +46384.736}
SPL {X  -159.990, Y  +674.512, Z    +0.000, E1    -0.026, E3 +46384.800}
SPL {X  -159.990, Y  +672.767, Z    +0.000, E1    +3.705, E3 +46384.814}
SPL {X  -159.990, Y  +669.310, Z    +0.000, E1   +12.444, E3 +46384.887}
SPL {X  -159.990, Y  +665.511, Z    +0.000, E1   +22.359, E3 +46385.046}
SPL {X  -159.990, Y  +658.432, Z    +0.000, E1   +38.720, E3 +46385.571}
SPL {X  -159.990, Y  +646.280, Z    +0.000, E1   +56.156, E3 +46387.100}
SPL {X  -159.990, Y  +625.549, Z    +0.000, E1   +67.208, E3 +46391.621}
SPL {X  -159.990, Y  +550.186, Z    +0.000, E1   +73.637, E3 +46417.027}
SPL {X  -159.878, Y  +371.520, Z    +0.000, E1   +74.559, E3 +46499.789}
SPL {X  -159.109, Y  +360.737, Z    +0.000, E1   +74.490, E3 +46506.913}
SPL {X  -156.915, Y  +346.281, Z    +0.000, E1   +74.304, E3 +46517.616}
ENDSPLINE

SPLINE
SPL {X  -159.697, Y  +367.814, Z    +0.000, E1   +71.217, E3 +46534.935}
ENDSPLINE

SPLINE
SPL {X  -156.028, Y  +342.114, Z    +0.000, E1   +72.020, E3 +46545.088}
SPL {X  -150.925, Y  +324.412, Z    +0.000, E1   +72.419, E3 +46552.881}
SPL {X  -144.972, Y  +309.824, Z    +0.000, E1   +72.799, E3 +46558.483}
SPL {X  -139.605, Y  +299.351, Z    +0.000, E1   +73.035, E3 +46562.615}
SPL {X  -136.475, Y  +294.006, Z    +0.000, E1   +72.670, E3 +46568.400}
SPL {X  -133.214, Y  +288.895, Z    +0.000, E1   +72.272, E3 +46574.047}
SPL {X  -129.829, Y  +284.006, Z    +0.000, E1   +71.844, E3 +46579.522}
SPL {X  -125.428, Y  +278.179, Z    +0.000, E1   +71.273, E3 +46586.060}
SPL {X  -120.729, Y  +272.518, Z    +0.000, E1   +70.593, E3 +46592.369}
SPL {X   -77.409, Y  +237.483, Z    +0.000, E1   +59.013, E3 +46687.220}
ENDSPLINE

SPLINE
SPL {X  -103.775, Y  +255.731, Z    +0.000, E1   +56.205, E3 +46883.933}
SPL {X  -141.196, Y  +302.265, Z    +0.000, E1   +49.914, E3 +46921.418}
SPL {X  -153.296, Y  +331.706, Z    +0.000, E1   +38.681, E3 +46929.838}
SPL {X  -157.534, Y  +349.577, Z    +0.000, E1   +27.748, E3 +46932.465}
SPL {X  -159.460, Y  +364.489, Z    +0.000, E1   +15.407, E3 +46933.761}
SPL {X  -159.962, Y  +374.520, Z    +0.000, E1    +5.534, E3 +46934.156}
SPL {X  -159.990, Y  +379.490, Z    +0.000, E1    +0.023, E3 +46934.214}
SPL {X  -159.990, Y  +381.667, Z    +0.000, E1    -4.707, E3 +46934.236}
SPL {X  -159.990, Y  +385.814, Z    +0.000, E1   -15.621, E3 +46934.340}
SPL {X  -159.990, Y  +390.948, Z    +0.000, E1   -28.850, E3 +46934.616}
SPL {X  -159.990, Y  +399.006, Z    +0.000, E1   -45.565, E3 +46935.328}
SPL {X  -159.990, Y  +410.008, Z    +0.000, E1   -58.546, E3 +46936.938}
SPL {X  -159.990, Y  +430.714, Z    +0.000, E1   -67.965, E3 +46941.743}
SPL {X  -159.990, Y  +500.758, Z    +0.000, E1   -73.927, E3 +46964.419}
SPL {X  -158.798, Y  +695.991, Z    +0.000, E1   -74.986, E3 +47052.256}
SPL {X  -156.512, Y  +709.677, Z    +0.000, E1   -74.772, E3 +47062.399}
SPL {X  -153.684, Y  +720.975, Z    +0.000, E1   -74.508, E3 +47071.687}
SPL {X  -150.879, Y  +729.719, Z    +0.000, E1   -74.224, E3 +47079.481}
SPL {X  -148.237, Y  +736.689, Z    +0.000, E1   -73.960, E3 +47086.035}
SPL {X  -145.190, Y  +743.705, Z    +0.000, E1   -73.640, E3 +47092.956}
SPL {X  -141.940, Y  +750.322, Z    +0.000, E1   -73.290, E3 +47099.722}
SPL {X  -138.555, Y  +756.496, Z    +0.000, E1   -72.905, E3 +47106.287}
SPL {X  -135.025, Y  +762.319, Z    +0.000, E1   -72.483, E3 +47112.667}
SPL {X  -131.747, Y  +767.272, Z    +0.000, E1   -72.071, E3 +47118.192}
SPL {X  -127.432, Y  +773.236, Z    +0.000, E1   -71.530, E3 +47124.877}
SPL {X  -124.036, Y  +777.554, Z    +0.000, E1   -71.026, E3 +47129.776}
SPL {X  -120.782, Y  +781.422, Z    +0.000, E1   -70.584, E3 +47134.034}
SPL {X   -74.295, Y  +818.193, Z    +0.000, E1   -57.793, E3 +47244.364}
ENDSPLINE

SPLINE
SPL {X  -120.240, Y  +782.043, Z    +0.000, E1   -55.019, E3 +47442.860}
SPL {X  -145.777, Y  +742.423, Z    +0.000, E1   -46.722, E3 +47464.739}
SPL {X  -154.920, Y  +716.458, Z    +0.000, E1   -35.175, E3 +47470.794}
SPL {X  -158.252, Y  +700.019, Z    +0.000, E1   -24.087, E3 +47473.046}
SPL {X  -159.676, Y  +686.525, Z    +0.000, E1   -12.514, E3 +47474.036}
SPL {X  -159.990, Y  +674.678, Z    +0.000, E1    -0.382, E3 +47474.351}
SPL {X  -159.990, Y  +672.767, Z    +0.000, E1    +3.705, E3 +47474.366}
SPL {X  -159.990, Y  +669.310, Z    +0.000, E1   +12.444, E3 +47474.440}
SPL {X  -159.990, Y  +665.511, Z    +0.000, E1   +22.359, E3 +47474.598}
SPL {X  -159.990, Y  +660.776, Z    +0.000, E1   +34.018, E3 +47474.905}
SPL {X  -159.990, Y  +655.863, Z    +0.000, E1   +43.768, E3 +47475.362}
SPL {X  -159.990, Y  +646.280, Z    +0.000, E1   +56.156, E3 +47476.652}
SPL {X  -159.990, Y  +625.549, Z    +0.000, E1   +67.208, E3 +47481.173}
SPL {X  -159.990, Y  +550.186, Z    +0.000, E1   +73.637, E3 +47506.579}
SPL {X  -159.878, Y  +371.520, Z    +0.000, E1   +74.559, E3 +47589.341}
SPL {X  -159.109, Y  +360.737, Z    +0.000, E1   +74.490, E3 +47596.466}
SPL {X  -156.915, Y  +346.281, Z    +0.000, E1   +74.304, E3 +47607.169}
ENDSPLINE

SPLINE
SPL {X  -159.697, Y  +367.814, Z    +0.000, E1   +71.217, E3 +47624.487}
ENDSPLINE

SPLINE
SPL {X  -157.536, Y  +349.586, Z    +0.000, E1   +71.787, E3 +47631.785}
SPL {X  -154.855, Y  +337.291, Z    +0.000, E1   +72.155, E3 +47636.539}
SPL {X  -150.925, Y  +324.412, Z    +0.000, E1   +72.419, E3 +47642.433}
SPL {X  -144.972, Y  +309.824, Z    +0.000, E1   +72.799, E3 +47648.035}
SPL {X  -139.605, Y  +299.351, Z    +0.000, E1   +73.035, E3 +47652.167}
SPL {X  -136.475, Y  +294.006, Z    +0.000, E1   +72.670, E3 +47657.952}
SPL {X  -133.214, Y  +288.895, Z    +0.000, E1   +72.272, E3 +47663.600}
SPL {X  -129.829, Y  +284.006, Z    +0.000, E1   +71.844, E3 +47669.075}
SPL {X  -126.314, Y  +279.309, Z    +0.000, E1   +71.374, E3 +47674.367}
SPL {X  -122.705, Y  +274.834, Z    +0.000, E1   +70.869, E3 +47679.378}
SPL {X  -119.804, Y  +271.463, Z    +0.000, E1   +70.429, E3 +47683.097}
SPL {X   -77.409, Y  +237.483, Z    +0.000, E1   +59.013, E3 +47776.772}
ENDSPLINE

SPLINE
SPL {X  -103.775, Y  +255.731, Z    +0.000, E1   +56.205, E3 +47973.486}
SPL {X  -141.196, Y  +302.265, Z    +0.000, E1   +49.914, E3 +48010.971}
SPL {X  -155.405, Y  +339.473, Z    +0.000, E1   +34.418, E3 +48020.671}
SPL {X  -158.399, Y  +354.990, Z    +0.000, E1   +23.559, E3 +48022.603}
SPL {X  -159.460, Y  +364.489, Z    +0.000, E1   +15.407, E3 +48023.313}
SPL {X  -159.962, Y  +374.520, Z    +0.000, E1    +5.534, E3 +48023.709}
SPL {X  -159.990, Y  +379.490, Z    +0.000, E1    +0.023, E3 +48023.766}
SPL {X  -159.990, Y  +381.667, Z    +0.000, E1    -4.707, E3 +48023.788}
SPL {X  -159.990, Y  +385.814, Z    +0.000, E1   -15.621, E3 +48023.892}
SPL {X  -159.990, Y  +390.948, Z    +0.000, E1   -28.850, E3 +48024.168}
SPL {X  -159.990, Y  +399.006, Z    +0.000, E1   -45.565, E3 +48024.880}
SPL {X  -159.990, Y  +410.008, Z    +0.000, E1   -58.546, E3 +48026.490}
SPL {X  -159.990, Y  +426.664, Z    +0.000, E1   -66.963, E3 +48030.111}
SPL {X  -159.990, Y  +494.829, Z    +0.000, E1   -73.764, E3 +48051.875}
SPL {X  -158.798, Y  +695.991, Z    +0.000, E1   -74.986, E3 +48141.808}
SPL {X  -156.512, Y  +709.677, Z    +0.000, E1   -74.772, E3 +48151.952}
SPL {X  -153.684, Y  +720.975, Z    +0.000, E1   -74.508, E3 +48161.239}
SPL {X  -149.353, Y  +733.863, Z    +0.000, E1   -74.100, E3 +48172.827}
SPL {X  -145.190, Y  +743.705, Z    +0.000, E1   -73.640, E3 +48182.508}
SPL {X  -141.940, Y  +750.322, Z    +0.000, E1   -73.290, E3 +48189.275}
SPL {X  -138.555, Y  +756.496, Z    +0.000, E1   -72.905, E3 +48195.840}
SPL {X  -135.025, Y  +762.319, Z    +0.000, E1   -72.483, E3 +48202.219}
SPL {X  -131.747, Y  +767.272, Z    +0.000, E1   -72.071, E3 +48207.744}
SPL {X  -128.648, Y  +771.613, Z    +0.000, E1   -71.666, E3 +48212.636}
SPL {X  -125.012, Y  +776.344, Z    +0.000, E1   -71.184, E3 +48217.948}
SPL {X  -120.782, Y  +781.422, Z    +0.000, E1   -70.584, E3 +48223.586}
SPL {X   -74.295, Y  +818.193, Z    +0.000, E1   -57.793, E3 +48333.917}
ENDSPLINE

SPLINE
SPL {X  -120.240, Y  +782.043, Z    +0.000, E1   -55.019, E3 +48532.412}
SPL {X  -145.777, Y  +742.423, Z    +0.000, E1   -46.722, E3 +48554.292}
SPL {X  -154.920, Y  +716.458, Z    +0.000, E1   -35.175, E3 +48560.347}
SPL {X  -159.063, Y  +693.702, Z    +0.000, E1   -19.028, E3 +48563.128}
SPL {X  -159.958, Y  +679.684, Z    +0.000, E1    -5.688, E3 +48563.840}
SPL {X  -159.990, Y  +674.512, Z    +0.000, E1    -0.026, E3 +48563.905}
SPL {X  -159.990, Y  +672.767, Z    +0.000, E1    +3.705, E3 +48563.918}
SPL {X  -159.990, Y  +669.310, Z    +0.000, E1   +12.444, E3 +48563.992}
SPL {X  -159.990, Y  +665.511, Z    +0.000, E1   +22.359, E3 +48564.151}
SPL {X  -159.990, Y  +658.432, Z    +0.000, E1   +38.720, E3 +48564.676}
SPL {X  -159.990, Y  +646.280, Z    +0.000, E1   +56.156, E3 +48566.204}
SPL {X  -159.990, Y  +625.549, Z    +0.000, E1   +67.208, E3 +48570.726}
SPL {X  -159.990, Y  +550.186, Z    +0.000, E1   +73.637, E3 +48596.131}
SPL {X  -159.493, Y  +364.902, Z    +0.000, E1   +74.541, E3 +48683.125}
SPL {X  -156.915, Y  +346.281, Z    +0.000, E1   +74.304, E3 +48696.721}
ENDSPLINE

SPLINE
SPL {X  -159.697, Y  +367.814, Z    +0.000, E1   +71.217, E3 +48714.039}
ENDSPLINE

SPLINE
SPL {X  -157.536, Y  +349.586, Z    +0.000, E1   +71.787, E3 +48721.337}
SPL {X  -154.855, Y  +337.291, Z    +0.000, E1   +72.155, E3 +48726.091}
SPL {X  -150.925, Y  +324.412, Z    +0.000, E1   +72.419, E3 +48731.986}
SPL {X  -144.972, Y  +309.824, Z    +0.000, E1   +72.799, E3 +48737.588}
SPL {X  -139.605, Y  +299.351, Z    +0.000, E1   +73.035, E3 +48741.719}
SPL {X  -136.475, Y  +294.006, Z    +0.000, E1   +72.670, E3 +48747.504}
SPL {X  -133.214, Y  +288.895, Z    +0.000, E1   +72.272, E3 +48753.152}
SPL {X  -129.829, Y  +284.006, Z    +0.000, E1   +71.844, E3 +48758.627}
SPL {X  -125.428, Y  +278.179, Z    +0.000, E1   +71.273, E3 +48765.164}
SPL {X  -120.729, Y  +272.518, Z    +0.000, E1   +70.593, E3 +48771.474}
SPL {X   -77.409, Y  +237.483, Z    +0.000, E1   +59.013, E3 +48866.325}
ENDSPLINE

SPLINE
SPL {X  -103.775, Y  +255.731, Z    +0.000, E1   +56.205, E3 +49063.038}
SPL {X  -141.196, Y  +302.265, Z    +0.000, E1   +49.914, E3 +49100.523}
SPL {X  -155.405, Y  +339.473, Z    +0.000, E1   +34.418, E3 +49110.223}
SPL {X  -159.172, Y  +361.346, Z    +0.000, E1   +18.323, E3 +49112.648}
SPL {X  -159.962, Y  +374.520, Z    +0.000, E1    +5.534, E3 +49113.261}
SPL {X  -159.990, Y  +379.490, Z    +0.000, E1    +0.023, E3 +49113.318}
SPL {X  -159.990, Y  +381.667, Z    +0.000, E1    -4.707, E3 +49113.340}
SPL {X  -159.990, Y  +385.814, Z    +0.000, E1   -15.621, E3 +49113.444}
SPL {X  -159.990, Y  +390.948, Z    +0.000, E1   -28.850, E3 +49113.720}
SPL {X  -159.990, Y  +399.006, Z    +0.000, E1   -45.565, E3 +49114.432}
SPL {X  -159.990, Y  +410.008, Z    +0.000, E1   -58.546, E3 +49116.042}
SPL {X  -159.990, Y  +426.664, Z    +0.000, E1   -66.963, E3 +49119.663}
SPL {X  -159.990, Y  +494.829, Z    +0.000, E1   -73.764, E3 +49141.428}
SPL {X  -158.798, Y  +695.991, Z    +0.000, E1   -74.986, E3 +49231.360}
SPL {X  -156.512, Y  +709.677, Z    +0.000, E1   -74.772, E3 +49241.504}
SPL {X  -153.684, Y  +720.975, Z    +0.000, E1   -74.508, E3 +49250.791}
SPL {X  -149.353, Y  +733.863, Z    +0.000, E1   -74.100, E3 +49262.379}
SPL {X  -145.190, Y  +743.705, Z    +0.000, E1   -73.640, E3 +49272.060}
SPL {X  -141.940, Y  +750.322, Z    +0.000, E1   -73.290, E3 +49278.827}
SPL {X  -138.555, Y  +756.496, Z    +0.000, E1   -72.905, E3 +49285.392}
SPL {X  -135.025, Y  +762.319, Z    +0.000, E1   -72.483, E3 +49291.771}
SPL {X  -131.747, Y  +767.272, Z    +0.000, E1   -72.071, E3 +49297.296}
SPL {X  -128.648, Y  +771.613, Z    +0.000, E1   -71.666, E3 +49302.189}
SPL {X  -125.012, Y  +776.344, Z    +0.000, E1   -71.184, E3 +49307.500}
SPL {X  -121.578, Y  +780.498, Z    +0.000, E1   -70.681, E3 +49312.144}
SPL {X  -119.460, Y  +782.925, Z    +0.000, E1   -70.353, E3 +49314.808}
SPL {X   -74.295, Y  +818.193, Z    +0.000, E1   -57.793, E3 +49423.469}
ENDSPLINE

SPLINE
SPL {X  -120.240, Y  +782.043, Z    +0.000, E1   -55.019, E3 +49621.965}
SPL {X  -145.777, Y  +742.423, Z    +0.000, E1   -46.722, E3 +49643.844}
SPL {X  -154.920, Y  +716.458, Z    +0.000, E1   -35.175, E3 +49649.899}
SPL {X  -159.063, Y  +693.702, Z    +0.000, E1   -19.028, E3 +49652.680}
SPL {X  -159.958, Y  +679.684, Z    +0.000, E1    -5.688, E3 +49653.392}
SPL {X  -159.990, Y  +674.512, Z    +0.000, E1    -0.026, E3 +49653.457}
SPL {X  -159.990, Y  +672.767, Z    +0.000, E1    +3.705, E3 +49653.470}
SPL {X  -159.990, Y  +669.310, Z    +0.000, E1   +12.444, E3 +49653.544}
SPL {X  -159.990, Y  +665.511, Z    +0.000, E1   +22.359, E3 +49653.703}
SPL {X  -159.990, Y  +660.776, Z    +0.000, E1   +34.018, E3 +49654.010}
SPL {X  -159.990, Y  +655.863, Z    +0.000, E1   +43.768, E3 +49654.467}
SPL {X  -159.990, Y  +646.280, Z    +0.000, E1   +56.156, E3 +49655.756}
SPL {X  -159.990, Y  +625.549, Z    +0.000, E1   +67.208, E3 +49660.278}
SPL {X  -159.990, Y  +550.186, Z    +0.000, E1   +73.637, E3 +49685.684}
SPL {X  -159.493, Y  +364.902, Z    +0.000, E1   +74.541, E3 +49772.677}
SPL {X  -156.915, Y  +346.281, Z    +0.000, E1   +74.304, E3 +49786.273}
ENDSPLINE

SPLINE
SPL {X  -159.697, Y  +367.814, Z    +0.000, E1   +71.217, E3 +49803.592}
ENDSPLINE

SPLINE
SPL {X  -156.028, Y  +342.114, Z    +0.000, E1   +72.020, E3 +49813.745}
SPL {X  -150.925, Y  +324.412, Z    +0.000, E1   +72.419, E3 +49821.538}
SPL {X  -144.972, Y  +309.824, Z    +0.000, E1   +72.799, E3 +49827.140}
SPL {X  -139.605, Y  +299.351, Z    +0.000, E1   +73.035, E3 +49831.271}
SPL {X  -136.475, Y  +294.006, Z    +0.000, E1   +72.670, E3 +49837.056}
SPL {X  -133.214, Y  +288.895, Z    +0.000, E1   +72.272, E3 +49842.704}
SPL {X  -129.829, Y  +284.006, Z    +0.000, E1   +71.844, E3 +49848.179}
SPL {X  -125.428, Y  +278.179, Z    +0.000, E1   +71.273, E3 +49854.717}
SPL {X  -120.729, Y  +272.518, Z    +0.000, E1   +70.593, E3 +49861.026}
SPL {X   -77.409, Y  +237.483, Z    +0.000, E1   +59.013, E3 +49955.877}
ENDSPLINE

SPLINE
SPL {X  -103.775, Y  +255.731, Z    +0.000, E1   +56.205, E3 +50152.590}
SPL {X  -141.196, Y  +302.265, Z    +0.000, E1   +49.914, E3 +50190.075}
SPL {X  -153.296, Y  +331.706, Z    +0.000, E1   +38.681, E3 +50198.494}
SPL {X  -157.534, Y  +349.577, Z    +0.000, E1   +27.748, E3 +50201.122}
SPL {X  -159.460, Y  +364.489, Z    +0.000, E1   +15.407, E3 +50202.417}
SPL {X  -159.962, Y  +374.520, Z    +0.000, E1    +5.534, E3 +50202.813}
SPL {X  -159.990, Y  +379.490, Z    +0.000, E1    +0.023, E3 +50202.871}
SPL {X  -159.990, Y  +381.667, Z    +0.000, E1    -4.707, E3 +50202.893}
SPL {X  -159.990, Y  +387.434, Z    +0.000, E1   -19.600, E3 +50203.075}
SPL {X  -159.990, Y  +392.971, Z    +0.000, E1   -33.903, E3 +50203.408}
SPL {X  -159.990, Y  +399.006, Z    +0.000, E1   -45.565, E3 +50203.984}
SPL {X  -159.990, Y  +410.008, Z    +0.000, E1   -58.546, E3 +50205.595}
SPL {X  -159.990, Y  +426.664, Z    +0.000, E1   -66.963, E3 +50209.216}
SPL {X  -159.990, Y  +494.829, Z    +0.000, E1   -73.764, E3 +50230.980}
SPL {X  -158.798, Y  +695.991, Z    +0.000, E1   -74.986, E3 +50320.913}
SPL {X  -156.512, Y  +709.677, Z    +0.000, E1   -74.772, E3 +50331.056}
SPL {X  -153.684, Y  +720.975, Z    +0.000, E1   -74.508, E3 +50340.343}
SPL {X  -149.353, Y  +733.863, Z    +0.000, E1   -74.100, E3 +50351.931}
SPL {X  -145.190, Y  +743.705, Z    +0.000, E1   -73.640, E3 +50361.612}
SPL {X  -141.940, Y  +750.322, Z    +0.000, E1   -73.290, E3 +50368.379}
SPL {X  -138.555, Y  +756.496, Z    +0.000, E1   -72.905, E3 +50374.944}
SPL {X  -135.025, Y  +762.319, Z    +0.000, E1   -72.483, E3 +50381.324}
SPL {X  -131.747, Y  +767.272, Z    +0.000, E1   -72.071, E3 +50386.849}
SPL {X  -127.432, Y  +773.236, Z    +0.000, E1   -71.530, E3 +50393.534}
SPL {X  -124.036, Y  +777.554, Z    +0.000, E1   -71.026, E3 +50398.432}
SPL {X  -120.782, Y  +781.422, Z    +0.000, E1   -70.584, E3 +50402.690}
SPL {X   -74.295, Y  +818.193, Z    +0.000, E1   -57.793, E3 +50513.021}
ENDSPLINE

SPLINE
SPL {X  -105.102, Y  +797.125, Z    +0.000, E1   -55.734, E3 +50692.388}
SPL {X  -126.361, Y  +774.631, Z    +0.000, E1   -54.192, E3 +50718.055}
SPL {X  -145.777, Y  +742.423, Z    +0.000, E1   -46.722, E3 +50733.396}
SPL {X  -154.920, Y  +716.458, Z    +0.000, E1   -35.175, E3 +50739.451}
SPL {X  -158.252, Y  +700.019, Z    +0.000, E1   -24.087, E3 +50741.703}
SPL {X  -159.676, Y  +686.525, Z    +0.000, E1   -12.514, E3 +50742.693}
SPL {X  -159.990, Y  +674.678, Z    +0.000, E1    -0.382, E3 +50743.008}
SPL {X  -159.990, Y  +672.767, Z    +0.000, E1    +3.705, E3 +50743.022}
SPL {X  -159.990, Y  +669.310, Z    +0.000, E1   +12.444, E3 +50743.096}
SPL {X  -159.990, Y  +665.511, Z    +0.000, E1   +22.359, E3 +50743.255}
SPL {X  -159.990, Y  +658.432, Z    +0.000, E1   +38.720, E3 +50743.780}
SPL {X  -159.990, Y  +646.280, Z    +0.000, E1   +56.156, E3 +50745.309}
SPL {X  -159.990, Y  +625.549, Z    +0.000, E1   +67.208, E3 +50749.830}
SPL {X  -159.990, Y  +550.186, Z    +0.000, E1   +73.637, E3 +50775.236}
SPL {X  -159.878, Y  +371.520, Z    +0.000, E1   +74.559, E3 +50857.998}
SPL {X  -158.372, Y  +354.804, Z    +0.000, E1   +74.445, E3 +50869.303}
SPL {X  -156.009, Y  +342.031, Z    +0.000, E1   +74.195, E3 +50879.312}
ENDSPLINE

SPLINE
SPL {X  -159.697, Y  +367.814, Z    +0.000, E1   +71.217, E3 +50893.144}
ENDSPLINE

SPLINE
SPL {X  -156.028, Y  +342.114, Z    +0.000, E1   +72.020, E3 +50903.297}
SPL {X  -150.925, Y  +324.412, Z    +0.000, E1   +72.419, E3 +50911.090}
SPL {X  -144.972, Y  +309.824, Z    +0.000, E1   +72.799, E3 +50916.692}
SPL {X  -139.605, Y  +299.351, Z    +0.000, E1   +73.035, E3 +50920.824}
SPL {X  -136.475, Y  +294.006, Z    +0.000, E1   +72.670, E3 +50926.609}
SPL {X  -133.214, Y  +288.895, Z    +0.000, E1   +72.272, E3 +50932.256}
SPL {X  -129.829, Y  +284.006, Z    +0.000, E1   +71.844, E3 +50937.731}
SPL {X  -125.428, Y  +278.179, Z    +0.000, E1   +71.273, E3 +50944.269}
SPL {X  -120.729, Y  +272.518, Z    +0.000, E1   +70.593, E3 +50950.578}
SPL {X   -77.409, Y  +237.483, Z    +0.000, E1   +59.013, E3 +51045.429}
ENDSPLINE

SPLINE
SPL {X  -103.775, Y  +255.731, Z    +0.000, E1   +56.205, E3 +51242.142}
SPL {X  -133.021, Y  +288.605, Z    +0.000, E1   +53.007, E3 +51273.599}
SPL {X  -149.384, Y  +320.219, Z    +0.000, E1   +43.953, E3 +51285.322}
SPL {X  -157.534, Y  +349.577, Z    +0.000, E1   +27.748, E3 +51290.674}
SPL {X  -159.460, Y  +364.489, Z    +0.000, E1   +15.407, E3 +51291.970}
SPL {X  -159.962, Y  +374.520, Z    +0.000, E1    +5.534, E3 +51292.365}
SPL {X  -159.990, Y  +379.741, Z    +0.000, E1    -0.257, E3 +51292.424}
SPL {X  -159.990, Y  +384.604, Z    +0.000, E1   -12.124, E3 +51292.513}
SPL {X  -159.990, Y  +389.475, Z    +0.000, E1   -25.351, E3 +51292.726}
SPL {X  -159.990, Y  +395.000, Z    +0.000, E1   -38.121, E3 +51293.136}
SPL {X  -159.990, Y  +406.380, Z    +0.000, E1   -55.108, E3 +51294.578}
SPL {X  -159.990, Y  +426.664, Z    +0.000, E1   -66.963, E3 +51298.768}
SPL {X  -159.990, Y  +494.829, Z    +0.000, E1   -73.764, E3 +51320.532}
SPL {X  -158.798, Y  +695.991, Z    +0.000, E1   -74.986, E3 +51410.465}
SPL {X  -156.512, Y  +709.677, Z    +0.000, E1   -74.772, E3 +51420.608}
SPL {X  -153.684, Y  +720.975, Z    +0.000, E1   -74.508, E3 +51429.896}
SPL {X  -149.353, Y  +733.863, Z    +0.000, E1   -74.100, E3 +51441.483}
SPL {X  -145.190, Y  +743.705, Z    +0.000, E1   -73.640, E3 +51451.164}
SPL {X  -141.940, Y  +750.322, Z    +0.000, E1   -73.290, E3 +51457.931}
SPL {X  -138.555, Y  +756.496, Z    +0.000, E1   -72.905, E3 +51464.496}
SPL {X  -135.025, Y  +762.319, Z    +0.000, E1   -72.483, E3 +51470.876}
SPL {X  -131.747, Y  +767.272, Z    +0.000, E1   -72.071, E3 +51476.401}
SPL {X  -127.432, Y  +773.236, Z    +0.000, E1   -71.530, E3 +51483.086}
SPL {X  -124.036, Y  +777.554, Z    +0.000, E1   -71.026, E3 +51487.985}
SPL {X  -120.782, Y  +781.422, Z    +0.000, E1   -70.584, E3 +51492.243}
SPL {X   -74.295, Y  +818.193, Z    +0.000, E1   -57.793, E3 +51602.573}
ENDSPLINE

SPLINE
SPL {X  -120.240, Y  +782.043, Z    +0.000, E1   -55.019, E3 +51801.069}
SPL {X  -145.777, Y  +742.423, Z    +0.000, E1   -46.722, E3 +51822.948}
SPL {X  -154.920, Y  +716.458, Z    +0.000, E1   -35.175, E3 +51829.003}
SPL {X  -158.252, Y  +700.019, Z    +0.000, E1   -24.087, E3 +51831.255}
SPL {X  -159.676, Y  +686.525, Z    +0.000, E1   -12.514, E3 +51832.245}
SPL {X  -159.990, Y  +674.678, Z    +0.000, E1    -0.382, E3 +51832.560}
SPL {X  -159.990, Y  +672.767, Z    +0.000, E1    +3.705, E3 +51832.575}
SPL {X  -159.990, Y  +669.310, Z    +0.000, E1   +12.444, E3 +51832.649}
SPL {X  -159.990, Y  +665.511, Z    +0.000, E1   +22.359, E3 +51832.807}
SPL {X  -159.990, Y  +660.776, Z    +0.000, E1   +34.018, E3 +51833.114}
SPL {X  -159.990, Y  +655.863, Z    +0.000, E1   +43.768, E3 +51833.571}
SPL {X  -159.990, Y  +646.280, Z    +0.000, E1   +56.156, E3 +51834.861}
SPL {X  -159.990, Y  +625.549, Z    +0.000, E1   +67.208, E3 +51839.382}
SPL {X  -159.990, Y  +550.186, Z    +0.000, E1   +73.637, E3 +51864.788}
SPL {X  -159.878, Y  +371.520, Z    +0.000, E1   +74.559, E3 +51947.550}
SPL {X  -159.109, Y  +360.737, Z    +0.000, E1   +74.490, E3 +51954.674}
SPL {X  -156.915, Y  +346.281, Z    +0.000, E1   +74.304, E3 +51965.377}
ENDSPLINE

SPLINE
SPL {X  -159.697, Y  +367.814, Z    +0.000, E1   +71.217, E3 +51982.696}
ENDSPLINE

SPLINE
SPL {X  -156.028, Y  +342.114, Z    +0.000, E1   +72.020, E3 +51992.849}
SPL {X  -150.925, Y  +324.412, Z    +0.000, E1   +72.419, E3 +52000.642}
SPL {X  -146.819, Y  +313.931, Z    +0.000, E1   +72.621, E3 +52005.336}
SPL {X  -140.820, Y  +301.561, Z    +0.000, E1   +73.023, E3 +52009.252}
SPL {X  -136.475, Y  +294.006, Z    +0.000, E1   +72.670, E3 +52016.161}
SPL {X  -133.214, Y  +288.895, Z    +0.000, E1   +72.272, E3 +52021.809}
SPL {X  -129.829, Y  +284.006, Z    +0.000, E1   +71.844, E3 +52027.284}
SPL {X  -125.428, Y  +278.179, Z    +0.000, E1   +71.273, E3 +52033.821}
SPL {X  -120.729, Y  +272.518, Z    +0.000, E1   +70.593, E3 +52040.130}
SPL {X   -77.409, Y  +237.483, Z    +0.000, E1   +59.013, E3 +52134.981}
ENDSPLINE

